//     Enc/Inputs/In/nState1 @bit 1 <-> FB Inputs Channel 2/Status/Error
//     Enc/Inputs/In/nState1 @bit 1 <-> FB Inputs Channel 1/Status/Error
//     Enc/Inputs/In/nState1 @bit 14 <-> FB Inputs Channel 2/Status/Input cycle counter
//     Enc/Inputs/In/nState1 @bit 14 <-> FB Inputs Channel 1/Status/Input cycle counter
//     Enc/Inputs/In/nState1 @bit 2 <-> FB Inputs Channel 2/Status/Ready
//     Enc/Inputs/In/nState1 @bit 2 <-> FB Inputs Channel 1/Status/Ready
//     Enc/Inputs/In/nState1 @bit 13 <-> FB Inputs Channel 2/Status/TxPDO State
//     Enc/Inputs/In/nState1 @bit 13 <-> FB Inputs Channel 1/Status/TxPDO State
//     Enc/Inputs/In/nState1 <-> FB Inputs Channel 2/Status/Warning
//     Enc/Inputs/In/nState1 <-> FB Inputs Channel 1/Status/Warning
//   (this object) <-> PLC Rail (EtherCAT)/Power (EK1200)/Fiber Coupler (EK1521-0010)/Term 123 (EK1100)/Term 73 (EK1122)/PAX-DRL-02 (EK1100)/PAX-EL7047-E17
//     Drive/Inputs/In/nState1 @bit 3 <-> STM Status/Status/Error
//     Drive/Inputs/In/nState1 @bit 7 <-> STM Status/Status/Motor stall
//     Drive/Inputs/In/nState1 @bit 5 <-> STM Status/Status/Moving negative
//     Drive/Inputs/In/nState1 @bit 4 <-> STM Status/Status/Moving positive
//     Drive/Inputs/In/nState1 @bit 1 <-> STM Status/Status/Ready
//     Drive/Inputs/In/nState1 <-> STM Status/Status/Ready to enable
//     Drive/Inputs/In/nState1 @bit 6 <-> STM Status/Status/Torque reduced
//     Drive/Inputs/In/nState1 @bit 2 <-> STM Status/Status/Warning
//     Drive/Inputs/In/nState2 @bit 3 <-> STM Status/Status/Digital input 1
//     Drive/Inputs/In/nState2 @bit 4 <-> STM Status/Status/Digital input 2
//     Drive/Inputs/In/nState2 @bit 5 <-> STM Status/Status/Sync error
//     Drive/Inputs/In/nState2 @bit 7 <-> STM Status/Status/TxPDO Toggle
//     Drive/Inputs/In/nState4 @bit 1 <-> WcState/InputToggle
//     Drive/Inputs/In/nState4 <-> WcState/WcState
//     Drive/Outputs/Out/nCtrl1 <-> STM Control/Control/Enable
//     Drive/Outputs/Out/nCtrl1 @bit 2 <-> STM Control/Control/Reduce torque
//     Drive/Outputs/Out/nCtrl1 @bit 1 <-> STM Control/Control/Reset
//     Drive/Outputs/Out/nCtrl2 @bit 3 <-> STM Control/Control/Digital output 1
//     Drive/Outputs/Out/nDataOut2[0] <-> STM Velocity/Velocity
//   (this object) <-> PLC Rail (EtherCAT)/Power (EK1200)/Fiber Coupler (EK1521-0010)/Term 123 (EK1100)/Term 73 (EK1122)/PAX-DRL-02 (EK1100)/PAX-EL7047-E15
//     Drive/Inputs/In/nState1 @bit 3 <-> STM Status/Status/Error
//     Drive/Inputs/In/nState1 @bit 7 <-> STM Status/Status/Motor stall
//     Drive/Inputs/In/nState1 @bit 5 <-> STM Status/Status/Moving negative
//     Drive/Inputs/In/nState1 @bit 4 <-> STM Status/Status/Moving positive
//     Drive/Inputs/In/nState1 @bit 1 <-> STM Status/Status/Ready
//     Drive/Inputs/In/nState1 <-> STM Status/Status/Ready to enable
//     Drive/Inputs/In/nState1 @bit 6 <-> STM Status/Status/Torque reduced
//     Drive/Inputs/In/nState1 @bit 2 <-> STM Status/Status/Warning
//     Drive/Inputs/In/nState2 @bit 3 <-> STM Status/Status/Digital input 1
//     Drive/Inputs/In/nState2 @bit 4 <-> STM Status/Status/Digital input 2
//     Drive/Inputs/In/nState2 @bit 5 <-> STM Status/Status/Sync error
//     Drive/Inputs/In/nState2 @bit 7 <-> STM Status/Status/TxPDO Toggle
//     Drive/Inputs/In/nState4 @bit 1 <-> WcState/InputToggle
//     Drive/Inputs/In/nState4 <-> WcState/WcState
//     Drive/Outputs/Out/nCtrl1 <-> STM Control/Control/Enable
//     Drive/Outputs/Out/nCtrl1 @bit 2 <-> STM Control/Control/Reduce torque
//     Drive/Outputs/Out/nCtrl1 @bit 1 <-> STM Control/Control/Reset
//     Drive/Outputs/Out/nCtrl2 @bit 3 <-> STM Control/Control/Digital output 1
//     Drive/Outputs/Out/nDataOut2[0] <-> STM Velocity/Velocity
//   (this object) <-> PLC Rail (EtherCAT)/Power (EK1200)/Fiber Coupler (EK1521-0010)/Term 123 (EK1100)/Term 73 (EK1122)/PAX-DRL-02 (EK1100)/PAX-EL5042-E13
//     Enc/Inputs/In/nComState @bit 1 <-> WcState/InputToggle
//     Enc/Inputs/In/nComState <-> WcState/WcState
//     Enc/Inputs/In/nDataIn1 <-> FB Inputs Channel 1/Position
//     Enc/Inputs/In/nState1 @bit 12 <-> FB Inputs Channel 1/Status/Diag
//     Enc/Inputs/In/nState1 @bit 1 <-> FB Inputs Channel 1/Status/Error
//     Enc/Inputs/In/nState1 @bit 14 <-> FB Inputs Channel 1/Status/Input cycle counter
//     Enc/Inputs/In/nState1 @bit 2 <-> FB Inputs Channel 1/Status/Ready
//     Enc/Inputs/In/nState1 @bit 13 <-> FB Inputs Channel 1/Status/TxPDO State
//     Enc/Inputs/In/nState1 <-> FB Inputs Channel 1/Status/Warning
//   (this object) <-> PLC Rail (EtherCAT)/Power (EK1200)/Fiber Coupler (EK1521-0010)/Term 123 (EK1100)/Term 73 (EK1122)/PAX-DRL-02 (EK1100)/PAX-EL7047-E12
//     Drive/Inputs/In/nState1 @bit 3 <-> STM Status/Status/Error
//     Drive/Inputs/In/nState1 @bit 7 <-> STM Status/Status/Motor stall
//     Drive/Inputs/In/nState1 @bit 5 <-> STM Status/Status/Moving negative
//     Drive/Inputs/In/nState1 @bit 4 <-> STM Status/Status/Moving positive
//     Drive/Inputs/In/nState1 @bit 1 <-> STM Status/Status/Ready
//     Drive/Inputs/In/nState1 <-> STM Status/Status/Ready to enable
//     Drive/Inputs/In/nState1 @bit 6 <-> STM Status/Status/Torque reduced
//     Drive/Inputs/In/nState1 @bit 2 <-> STM Status/Status/Warning
//     Drive/Inputs/In/nState2 @bit 3 <-> STM Status/Status/Digital input 1
//     Drive/Inputs/In/nState2 @bit 4 <-> STM Status/Status/Digital input 2
//     Drive/Inputs/In/nState2 @bit 5 <-> STM Status/Status/Sync error
//     Drive/Inputs/In/nState2 @bit 7 <-> STM Status/Status/TxPDO Toggle
//     Drive/Inputs/In/nState4 @bit 1 <-> WcState/InputToggle
//     Drive/Inputs/In/nState4 <-> WcState/WcState
//     Drive/Outputs/Out/nCtrl1 <-> STM Control/Control/Enable
//     Drive/Outputs/Out/nCtrl1 @bit 2 <-> STM Control/Control/Reduce torque
//     Drive/Outputs/Out/nCtrl1 @bit 1 <-> STM Control/Control/Reset
//     Drive/Outputs/Out/nCtrl2 @bit 3 <-> STM Control/Control/Digital output 1
//     Drive/Outputs/Out/nDataOut2[0] <-> STM Velocity/Velocity
//   (this object) <-> PLC Rail (EtherCAT)/Power (EK1200)/Fiber Coupler (EK1521-0010)/Term 123 (EK1100)/Term 73 (EK1122)/PAX-DRL-02 (EK1100)/PAX-EL5042-E09
//     Enc/Inputs/In/nComState @bit 1 <-> WcState/InputToggle
//     Enc/Inputs/In/nComState <-> WcState/WcState
//     Enc/Inputs/In/nDataIn1 <-> FB Inputs Channel 2/Position
//     Enc/Inputs/In/nDataIn1 <-> FB Inputs Channel 1/Position
//     Enc/Inputs/In/nState1 @bit 12 <-> FB Inputs Channel 2/Status/Diag
//     Enc/Inputs/In/nState1 @bit 12 <-> FB Inputs Channel 1/Status/Diag
//     Enc/Inputs/In/nState1 @bit 1 <-> FB Inputs Channel 2/Status/Error
//     Enc/Inputs/In/nState1 @bit 1 <-> FB Inputs Channel 1/Status/Error
//     Enc/Inputs/In/nState1 @bit 14 <-> FB Inputs Channel 2/Status/Input cycle counter
//     Enc/Inputs/In/nState1 @bit 14 <-> FB Inputs Channel 1/Status/Input cycle counter
//     Enc/Inputs/In/nState1 @bit 2 <-> FB Inputs Channel 2/Status/Ready
//     Enc/Inputs/In/nState1 @bit 2 <-> FB Inputs Channel 1/Status/Ready
//     Enc/Inputs/In/nState1 @bit 13 <-> FB Inputs Channel 2/Status/TxPDO State
//     Enc/Inputs/In/nState1 @bit 13 <-> FB Inputs Channel 1/Status/TxPDO State
//     Enc/Inputs/In/nState1 <-> FB Inputs Channel 2/Status/Warning
//     Enc/Inputs/In/nState1 <-> FB Inputs Channel 1/Status/Warning
//   (this object) <-> PLC Rail (EtherCAT)/Power (EK1200)/Fiber Coupler (EK1521-0010)/Term 123 (EK1100)/Term 73 (EK1122)/PAX-DRL-02 (EK1100)/PAX-EL7047-E10
//     Drive/Inputs/In/nState1 @bit 3 <-> STM Status/Status/Error
//     Drive/Inputs/In/nState1 @bit 7 <-> STM Status/Status/Motor stall
//     Drive/Inputs/In/nState1 @bit 5 <-> STM Status/Status/Moving negative
//     Drive/Inputs/In/nState1 @bit 4 <-> STM Status/Status/Moving positive
//     Drive/Inputs/In/nState1 @bit 1 <-> STM Status/Status/Ready
//     Drive/Inputs/In/nState1 <-> STM Status/Status/Ready to enable
//     Drive/Inputs/In/nState1 @bit 6 <-> STM Status/Status/Torque reduced
//     Drive/Inputs/In/nState1 @bit 2 <-> STM Status/Status/Warning
//     Drive/Inputs/In/nState2 @bit 3 <-> STM Status/Status/Digital input 1
//     Drive/Inputs/In/nState2 @bit 4 <-> STM Status/Status/Digital input 2
//     Drive/Inputs/In/nState2 @bit 5 <-> STM Status/Status/Sync error
//     Drive/Inputs/In/nState2 @bit 7 <-> STM Status/Status/TxPDO Toggle
//     Drive/Inputs/In/nState4 @bit 1 <-> WcState/InputToggle
//     Drive/Inputs/In/nState4 <-> WcState/WcState
//     Drive/Outputs/Out/nCtrl1 <-> STM Control/Control/Enable
//     Drive/Outputs/Out/nCtrl1 @bit 2 <-> STM Control/Control/Reduce torque
//     Drive/Outputs/Out/nCtrl1 @bit 1 <-> STM Control/Control/Reset
//     Drive/Outputs/Out/nCtrl2 @bit 3 <-> STM Control/Control/Digital output 1
//     Drive/Outputs/Out/nDataOut2[0] <-> STM Velocity/Velocity
//   (this object) <-> PLC Rail (EtherCAT)/Power (EK1200)/Fiber Coupler (EK1521-0010)/Term 123 (EK1100)/Term 73 (EK1122)/PAX-DRL-02 (EK1100)/PAX-EL7047-E08
//     Drive/Inputs/In/nState1 @bit 3 <-> STM Status/Status/Error
//     Drive/Inputs/In/nState1 @bit 7 <-> STM Status/Status/Motor stall
//     Drive/Inputs/In/nState1 @bit 5 <-> STM Status/Status/Moving negative
//     Drive/Inputs/In/nState1 @bit 4 <-> STM Status/Status/Moving positive
//     Drive/Inputs/In/nState1 @bit 1 <-> STM Status/Status/Ready
//     Drive/Inputs/In/nState1 <-> STM Status/Status/Ready to enable
//     Drive/Inputs/In/nState1 @bit 6 <-> STM Status/Status/Torque reduced
//     Drive/Inputs/In/nState1 @bit 2 <-> STM Status/Status/Warning
//     Drive/Inputs/In/nState2 @bit 3 <-> STM Status/Status/Digital input 1
//     Drive/Inputs/In/nState2 @bit 4 <-> STM Status/Status/Digital input 2
//     Drive/Inputs/In/nState2 @bit 5 <-> STM Status/Status/Sync error
//     Drive/Inputs/In/nState2 @bit 7 <-> STM Status/Status/TxPDO Toggle
//     Drive/Inputs/In/nState4 @bit 1 <-> WcState/InputToggle
//     Drive/Inputs/In/nState4 <-> WcState/WcState
//     Drive/Outputs/Out/nCtrl1 <-> STM Control/Control/Enable
//     Drive/Outputs/Out/nCtrl1 @bit 2 <-> STM Control/Control/Reduce torque
//     Drive/Outputs/Out/nCtrl1 @bit 1 <-> STM Control/Control/Reset
//     Drive/Outputs/Out/nCtrl2 @bit 3 <-> STM Control/Control/Digital output 1
//     Drive/Outputs/Out/nDataOut2[0] <-> STM Velocity/Velocity
//   (this object) <-> PLC Rail (EtherCAT)/Power (EK1200)/Fiber Coupler (EK1521-0010)/Term 123 (EK1100)/Term 73 (EK1122)/PAX-DRL-02 (EK1100)/PAX-EL5042-E05
//     Enc/Inputs/In/nComState @bit 1 <-> WcState/InputToggle
//     Enc/Inputs/In/nComState <-> WcState/WcState
//     Enc/Inputs/In/nDataIn1 <-> FB Inputs Channel 2/Position
//     Enc/Inputs/In/nDataIn1 <-> FB Inputs Channel 1/Position
//     Enc/Inputs/In/nState1 @bit 12 <-> FB Inputs Channel 2/Status/Diag
//     Enc/Inputs/In/nState1 @bit 12 <-> FB Inputs Channel 1/Status/Diag
//     Enc/Inputs/In/nState1 @bit 1 <-> FB Inputs Channel 2/Status/Error
//     Enc/Inputs/In/nState1 @bit 1 <-> FB Inputs Channel 1/Status/Error
//     Enc/Inputs/In/nState1 @bit 14 <-> FB Inputs Channel 2/Status/Input cycle counter
//     Enc/Inputs/In/nState1 @bit 14 <-> FB Inputs Channel 1/Status/Input cycle counter
//     Enc/Inputs/In/nState1 @bit 2 <-> FB Inputs Channel 2/Status/Ready
//     Enc/Inputs/In/nState1 @bit 2 <-> FB Inputs Channel 1/Status/Ready
//     Enc/Inputs/In/nState1 @bit 13 <-> FB Inputs Channel 2/Status/TxPDO State
//     Enc/Inputs/In/nState1 @bit 13 <-> FB Inputs Channel 1/Status/TxPDO State
//     Enc/Inputs/In/nState1 <-> FB Inputs Channel 2/Status/Warning
//     Enc/Inputs/In/nState1 <-> FB Inputs Channel 1/Status/Warning
//   (this object) <-> PLC Rail (EtherCAT)/Power (EK1200)/Fiber Coupler (EK1521-0010)/Term 123 (EK1100)/Term 73 (EK1122)/PAX-DRL-02 (EK1100)/PAX-EL7047-E06
//     Drive/Inputs/In/nState1 @bit 3 <-> STM Status/Status/Error
//     Drive/Inputs/In/nState1 @bit 7 <-> STM Status/Status/Motor stall
//     Drive/Inputs/In/nState1 @bit 5 <-> STM Status/Status/Moving negative
//     Drive/Inputs/In/nState1 @bit 4 <-> STM Status/Status/Moving positive
//     Drive/Inputs/In/nState1 @bit 1 <-> STM Status/Status/Ready
//     Drive/Inputs/In/nState1 <-> STM Status/Status/Ready to enable
//     Drive/Inputs/In/nState1 @bit 6 <-> STM Status/Status/Torque reduced
//     Drive/Inputs/In/nState1 @bit 2 <-> STM Status/Status/Warning
//     Drive/Inputs/In/nState2 @bit 3 <-> STM Status/Status/Digital input 1
//     Drive/Inputs/In/nState2 @bit 4 <-> STM Status/Status/Digital input 2
//     Drive/Inputs/In/nState2 @bit 5 <-> STM Status/Status/Sync error
//     Drive/Inputs/In/nState2 @bit 7 <-> STM Status/Status/TxPDO Toggle
//     Drive/Inputs/In/nState4 @bit 1 <-> WcState/InputToggle
//     Drive/Inputs/In/nState4 <-> WcState/WcState
//     Drive/Outputs/Out/nCtrl1 <-> STM Control/Control/Enable
//     Drive/Outputs/Out/nCtrl1 @bit 2 <-> STM Control/Control/Reduce torque
//     Drive/Outputs/Out/nCtrl1 @bit 1 <-> STM Control/Control/Reset
//     Drive/Outputs/Out/nCtrl2 @bit 3 <-> STM Control/Control/Digital output 1
//     Drive/Outputs/Out/nDataOut2[0] <-> STM Velocity/Velocity
//   (this object) <-> PLC Rail (EtherCAT)/Power (EK1200)/Fiber Coupler (EK1521-0010)/Term 123 (EK1100)/Term 73 (EK1122)/PAX-DRL-02 (EK1100)/PAX-EL7047-E04
//     Drive/Inputs/In/nState1 @bit 3 <-> STM Status/Status/Error
//     Drive/Inputs/In/nState1 @bit 7 <-> STM Status/Status/Motor stall
//     Drive/Inputs/In/nState1 @bit 5 <-> STM Status/Status/Moving negative
//     Drive/Inputs/In/nState1 @bit 4 <-> STM Status/Status/Moving positive
//     Drive/Inputs/In/nState1 @bit 1 <-> STM Status/Status/Ready
//     Drive/Inputs/In/nState1 <-> STM Status/Status/Ready to enable
//     Drive/Inputs/In/nState1 @bit 6 <-> STM Status/Status/Torque reduced
//     Drive/Inputs/In/nState1 @bit 2 <-> STM Status/Status/Warning
//     Drive/Inputs/In/nState2 @bit 3 <-> STM Status/Status/Digital input 1
//     Drive/Inputs/In/nState2 @bit 4 <-> STM Status/Status/Digital input 2
//     Drive/Inputs/In/nState2 @bit 5 <-> STM Status/Status/Sync error
//     Drive/Inputs/In/nState2 @bit 7 <-> STM Status/Status/TxPDO Toggle
//     Drive/Inputs/In/nState4 @bit 1 <-> WcState/InputToggle
//     Drive/Inputs/In/nState4 <-> WcState/WcState
//     Drive/Outputs/Out/nCtrl1 <-> STM Control/Control/Enable
//     Drive/Outputs/Out/nCtrl1 @bit 2 <-> STM Control/Control/Reduce torque
//     Drive/Outputs/Out/nCtrl1 @bit 1 <-> STM Control/Control/Reset
//     Drive/Outputs/Out/nCtrl2 @bit 3 <-> STM Control/Control/Digital output 1
//     Drive/Outputs/Out/nDataOut2[0] <-> STM Velocity/Velocity
//   (this object) <-> PLC Rail (EtherCAT)/Power (EK1200)/Fiber Coupler (EK1521-0010)/Term 123 (EK1100)/Term 73 (EK1122)/PAX-DRL-02 (EK1100)/PAX-EL5042-E02
//     Enc/Inputs/In/nComState @bit 1 <-> WcState/InputToggle
//     Enc/Inputs/In/nComState <-> WcState/WcState
//     Enc/Inputs/In/nDataIn1 <-> FB Inputs Channel 2/Position
//     Enc/Inputs/In/nDataIn1 <-> FB Inputs Channel 1/Position
//     Enc/Inputs/In/nState1 @bit 12 <-> FB Inputs Channel 2/Status/Diag
//     Enc/Inputs/In/nState1 @bit 12 <-> FB Inputs Channel 1/Status/Diag
//     Enc/Inputs/In/nState1 @bit 1 <-> FB Inputs Channel 2/Status/Error
//     Enc/Inputs/In/nState1 @bit 1 <-> FB Inputs Channel 1/Status/Error
//     Enc/Inputs/In/nState1 @bit 14 <-> FB Inputs Channel 2/Status/Input cycle counter
//     Enc/Inputs/In/nState1 @bit 14 <-> FB Inputs Channel 1/Status/Input cycle counter
//     Enc/Inputs/In/nState1 @bit 2 <-> FB Inputs Channel 2/Status/Ready
//     Enc/Inputs/In/nState1 @bit 2 <-> FB Inputs Channel 1/Status/Ready
//     Enc/Inputs/In/nState1 @bit 13 <-> FB Inputs Channel 2/Status/TxPDO State
//     Enc/Inputs/In/nState1 @bit 13 <-> FB Inputs Channel 1/Status/TxPDO State
//     Enc/Inputs/In/nState1 <-> FB Inputs Channel 2/Status/Warning
//     Enc/Inputs/In/nState1 <-> FB Inputs Channel 1/Status/Warning
//   (this object) <-> PLC Rail (EtherCAT)/Power (EK1200)/Fiber Coupler (EK1521-0010)/Term 123 (EK1100)/Term 73 (EK1122)/PAX-DRL-02 (EK1100)/PAX-EL7047-E03
//     Drive/Inputs/In/nState1 @bit 3 <-> STM Status/Status/Error
//     Drive/Inputs/In/nState1 @bit 7 <-> STM Status/Status/Motor stall
//     Drive/Inputs/In/nState1 @bit 5 <-> STM Status/Status/Moving negative
//     Drive/Inputs/In/nState1 @bit 4 <-> STM Status/Status/Moving positive
//     Drive/Inputs/In/nState1 @bit 1 <-> STM Status/Status/Ready
//     Drive/Inputs/In/nState1 <-> STM Status/Status/Ready to enable
//     Drive/Inputs/In/nState1 @bit 6 <-> STM Status/Status/Torque reduced
//     Drive/Inputs/In/nState1 @bit 2 <-> STM Status/Status/Warning
//     Drive/Inputs/In/nState2 @bit 3 <-> STM Status/Status/Digital input 1
//     Drive/Inputs/In/nState2 @bit 4 <-> STM Status/Status/Digital input 2
//     Drive/Inputs/In/nState2 @bit 5 <-> STM Status/Status/Sync error
//     Drive/Inputs/In/nState2 @bit 7 <-> STM Status/Status/TxPDO Toggle
//     Drive/Inputs/In/nState4 @bit 1 <-> WcState/InputToggle
//     Drive/Inputs/In/nState4 <-> WcState/WcState
//     Drive/Outputs/Out/nCtrl1 <-> STM Control/Control/Enable
//     Drive/Outputs/Out/nCtrl1 @bit 2 <-> STM Control/Control/Reduce torque
//     Drive/Outputs/Out/nCtrl1 @bit 1 <-> STM Control/Control/Reset
//     Drive/Outputs/Out/nCtrl2 @bit 3 <-> STM Control/Control/Digital output 1
//     Drive/Outputs/Out/nDataOut2[0] <-> STM Velocity/Velocity
//   (this object) <-> PLC Rail (EtherCAT)/Power (EK1200)/Fiber Coupler (EK1521-0010)/Term 123 (EK1100)/Term 73 (EK1122)/PAX-DRL-02 (EK1100)/PAX-EL7047-E01
//     Drive/Inputs/In/nState1 @bit 3 <-> STM Status/Status/Error
//     Drive/Inputs/In/nState1 @bit 7 <-> STM Status/Status/Motor stall
//     Drive/Inputs/In/nState1 @bit 5 <-> STM Status/Status/Moving negative
//     Drive/Inputs/In/nState1 @bit 4 <-> STM Status/Status/Moving positive
//     Drive/Inputs/In/nState1 @bit 1 <-> STM Status/Status/Ready
//     Drive/Inputs/In/nState1 <-> STM Status/Status/Ready to enable
//     Drive/Inputs/In/nState1 @bit 6 <-> STM Status/Status/Torque reduced
//     Drive/Inputs/In/nState1 @bit 2 <-> STM Status/Status/Warning
//     Drive/Inputs/In/nState2 @bit 3 <-> STM Status/Status/Digital input 1
//     Drive/Inputs/In/nState2 @bit 4 <-> STM Status/Status/Digital input 2
//     Drive/Inputs/In/nState2 @bit 5 <-> STM Status/Status/Sync error
//     Drive/Inputs/In/nState2 @bit 7 <-> STM Status/Status/TxPDO Toggle
//     Drive/Inputs/In/nState4 @bit 1 <-> WcState/InputToggle
//     Drive/Inputs/In/nState4 <-> WcState/WcState
//     Drive/Outputs/Out/nCtrl1 <-> STM Control/Control/Enable
//     Drive/Outputs/Out/nCtrl1 @bit 2 <-> STM Control/Control/Reduce torque
//     Drive/Outputs/Out/nCtrl1 @bit 1 <-> STM Control/Control/Reset
//     Drive/Outputs/Out/nCtrl2 @bit 3 <-> STM Control/Control/Digital output 1
//     Drive/Outputs/Out/nDataOut2[0] <-> STM Velocity/Velocity
//   kfe_rix_motion Instance <-> PLC Rail (EtherCAT)/EtherCAT Panel (EK1100)/EC E1 (EK1122)/X1 IM1K1-PPM (EK1100)/IM1K1-EL2004
//     PlcTask Outputs/Main.M1.bBrakeRelease <-> Channel 1/Output
//     PlcTask Outputs/PRG_IM1K1_PPM.fbIM1K1.fbGige.bGigePower <-> Channel 2/Output
//   kfe_rix_motion Instance <-> PLC Rail (EtherCAT)/EtherCAT Panel (EK1100)/EC E1 (EK1122)/X1 IM1K1-PPM (EK1100)/IM1K1-EL3062
//     PlcTask Inputs/PRG_IM1K1_PPM.fbIM1K1.fbPowerMeter.iVoltageINT <-> AI Standard Channel 1/Value
//   kfe_rix_motion Instance <-> PLC Rail (EtherCAT)/EtherCAT Panel (EK1100)/EC E1 (EK1122)/X1 IM1K1-PPM (EK1100)/IM1K1-EL3314
//     PlcTask Inputs/PRG_IM1K1_PPM.fbIM1K1.fbPowerMeter.fbTempSensor.bError <-> TC Inputs Channel 1/Status/Error
//     PlcTask Inputs/PRG_IM1K1_PPM.fbIM1K1.fbPowerMeter.fbTempSensor.bOverrange <-> TC Inputs Channel 1/Status/Overrange
//     PlcTask Inputs/PRG_IM1K1_PPM.fbIM1K1.fbPowerMeter.fbTempSensor.bUnderrange <-> TC Inputs Channel 1/Status/Underrange
//     PlcTask Inputs/PRG_IM1K1_PPM.fbIM1K1.fbPowerMeter.fbTempSensor.iRaw <-> TC Inputs Channel 1/Value
//     PlcTask Inputs/PRG_IM1K1_PPM.fbIM1K1.fbYagTempSensor.bError <-> TC Inputs Channel 2/Status/Error
//     PlcTask Inputs/PRG_IM1K1_PPM.fbIM1K1.fbYagTempSensor.bOverrange <-> TC Inputs Channel 2/Status/Overrange
//     PlcTask Inputs/PRG_IM1K1_PPM.fbIM1K1.fbYagTempSensor.bUnderrange <-> TC Inputs Channel 2/Status/Underrange
//     PlcTask Inputs/PRG_IM1K1_PPM.fbIM1K1.fbYagTempSensor.iRaw <-> TC Inputs Channel 2/Value
//   kfe_rix_motion Instance <-> PLC Rail (EtherCAT)/EtherCAT Panel (EK1100)/EC E1 (EK1122)/X1 IM1K1-PPM (EK1100)/IM1K1-EL4004
//     PlcTask Outputs/PRG_IM1K1_PPM.fbIM1K1.fbGige.iIlluminatorINT <-> AO Outputs Channel 1/Analog output
//   kfe_rix_motion Instance <-> PLC Rail (EtherCAT)/EtherCAT Panel (EK1100)/EC E1 (EK1122)/X1 IM1K1-PPM (EK1100)/IM1K1-EL7041
//     PlcTask Inputs/Main.M1.bLimitBackwardEnable <-> STM Status/Status/Digital input 2
//     PlcTask Inputs/Main.M1.bLimitForwardEnable <-> STM Status/Status/Digital input 1
//   kfe_rix_motion Instance <-> PLC Rail (EtherCAT)/EtherCAT Panel (EK1100)/EC E1 (EK1122)/X2 IM2K1-PPM (EK1100)/IM2K1-EL2004
//     PlcTask Outputs/Main.M2.bBrakeRelease <-> Channel 1/Output
//     PlcTask Outputs/PRG_IM2K1_PPM.fbIM2K1.fbGige.bGigePower <-> Channel 2/Output
//   kfe_rix_motion Instance <-> PLC Rail (EtherCAT)/EtherCAT Panel (EK1100)/EC E1 (EK1122)/X2 IM2K1-PPM (EK1100)/IM2K1-EL3062
//     PlcTask Inputs/PRG_IM2K1_PPM.fbIM2K1.fbPowerMeter.iVoltageINT <-> AI Standard Channel 1/Value
//   kfe_rix_motion Instance <-> PLC Rail (EtherCAT)/EtherCAT Panel (EK1100)/EC E1 (EK1122)/X2 IM2K1-PPM (EK1100)/IM2K1-EL3314
//     PlcTask Inputs/PRG_IM2K1_PPM.fbIM2K1.fbPowerMeter.fbTempSensor.bError <-> TC Inputs Channel 1/Status/Error
//     PlcTask Inputs/PRG_IM2K1_PPM.fbIM2K1.fbPowerMeter.fbTempSensor.bOverrange <-> TC Inputs Channel 1/Status/Overrange
//     PlcTask Inputs/PRG_IM2K1_PPM.fbIM2K1.fbPowerMeter.fbTempSensor.bUnderrange <-> TC Inputs Channel 1/Status/Underrange
//     PlcTask Inputs/PRG_IM2K1_PPM.fbIM2K1.fbPowerMeter.fbTempSensor.iRaw <-> TC Inputs Channel 1/Value
//     PlcTask Inputs/PRG_IM2K1_PPM.fbIM2K1.fbYagTempSensor.bError <-> TC Inputs Channel 2/Status/Error
//     PlcTask Inputs/PRG_IM2K1_PPM.fbIM2K1.fbYagTempSensor.bOverrange <-> TC Inputs Channel 2/Status/Overrange
//     PlcTask Inputs/PRG_IM2K1_PPM.fbIM2K1.fbYagTempSensor.bUnderrange <-> TC Inputs Channel 2/Status/Underrange
//     PlcTask Inputs/PRG_IM2K1_PPM.fbIM2K1.fbYagTempSensor.iRaw <-> TC Inputs Channel 2/Value
//   kfe_rix_motion Instance <-> PLC Rail (EtherCAT)/EtherCAT Panel (EK1100)/EC E1 (EK1122)/X2 IM2K1-PPM (EK1100)/IM2K1-EL4004
//     PlcTask Outputs/PRG_IM2K1_PPM.fbIM2K1.fbGige.iIlluminatorINT <-> AO Outputs Channel 1/Analog output
//   kfe_rix_motion Instance <-> PLC Rail (EtherCAT)/EtherCAT Panel (EK1100)/EC E1 (EK1122)/X2 IM2K1-PPM (EK1100)/IM2K1-EL7041
//     PlcTask Inputs/Main.M2.bLimitBackwardEnable <-> STM Status/Status/Digital input 2
//     PlcTask Inputs/Main.M2.bLimitForwardEnable <-> STM Status/Status/Digital input 1
//   kfe_rix_motion Instance <-> PLC Rail (EtherCAT)/Power (EK1200)/Fiber Coupler (EK1521-0010)/Term 123 (EK1100)/Term 124 (EK1122)/TM1K2-K2A (EK1100)/TM1K2-EL2004-E4
//     PlcTask Outputs/Main.M9.bBrakeRelease <-> Channel 1/Output
//   kfe_rix_motion Instance <-> PLC Rail (EtherCAT)/Power (EK1200)/Fiber Coupler (EK1521-0010)/Term 123 (EK1100)/Term 124 (EK1122)/TM1K2-K2A (EK1100)/TM1K2-EL3314-E5
//     PlcTask Inputs/PRG_TM1K2_ATM.fbTM1K2.fbThermoCouple1.bError <-> TC Inputs Channel 1/Status/Error
//     PlcTask Inputs/PRG_TM1K2_ATM.fbTM1K2.fbThermoCouple1.bOverrange <-> TC Inputs Channel 1/Status/Overrange
//     PlcTask Inputs/PRG_TM1K2_ATM.fbTM1K2.fbThermoCouple1.bUnderrange <-> TC Inputs Channel 1/Status/Underrange
//     PlcTask Inputs/PRG_TM1K2_ATM.fbTM1K2.fbThermoCouple1.iRaw <-> TC Inputs Channel 1/Value
//   kfe_rix_motion Instance <-> PLC Rail (EtherCAT)/Power (EK1200)/Fiber Coupler (EK1521-0010)/Term 123 (EK1100)/Term 124 (EK1122)/TM1K2-K2A (EK1100)/TM1K2-EL5042-E3
//     PlcTask Inputs/Main.M10.nRawEncoderULINT <-> FB Inputs Channel 2/Position
//     PlcTask Inputs/Main.M9.nRawEncoderULINT <-> FB Inputs Channel 1/Position
//   kfe_rix_motion Instance <-> PLC Rail (EtherCAT)/Power (EK1200)/Fiber Coupler (EK1521-0010)/Term 123 (EK1100)/Term 124 (EK1122)/TM1K2-K2A (EK1100)/TM1K2-EL7041-E1
//     PlcTask Inputs/Main.M9.bLimitBackwardEnable <-> STM Status/Status/Digital input 2
//     PlcTask Inputs/Main.M9.bLimitForwardEnable <-> STM Status/Status/Digital input 1
//   kfe_rix_motion Instance <-> PLC Rail (EtherCAT)/Power (EK1200)/Fiber Coupler (EK1521-0010)/Term 123 (EK1100)/Term 131 (EK1122)/LI2K2-K2A_OUT  (EK1100)/LI2K2-EL2004-E2
//     PlcTask Outputs/Main.M11.bBrakeRelease <-> Channel 1/Output
//   kfe_rix_motion Instance <-> PLC Rail (EtherCAT)/Power (EK1200)/Fiber Coupler (EK1521-0010)/Term 123 (EK1100)/Term 131 (EK1122)/LI2K2-K2A_OUT  (EK1100)/LI2K2-EL5042-E3
//     PlcTask Inputs/Main.M11.nRawEncoderULINT <-> FB Inputs Channel 1/Position
//   kfe_rix_motion Instance <-> PLC Rail (EtherCAT)/Power (EK1200)/Fiber Coupler (EK1521-0010)/Term 123 (EK1100)/Term 131 (EK1122)/LI2K2-K2A_OUT  (EK1100)/LI2K2-EL7041-E1
//     PlcTask Inputs/Main.M11.bLimitBackwardEnable <-> STM Status/Status/Digital input 2
//     PlcTask Inputs/Main.M11.bLimitForwardEnable <-> STM Status/Status/Digital input 1
//   kfe_rix_motion Instance <-> PLC Rail (EtherCAT)/Power (EK1200)/Fiber Coupler (EK1521-0010)/Term 123 (EK1100)/Term 131 (EK1122)/PF1K2-WFS (EK1100)/PF1K2-EL2004-E4
//     PlcTask Outputs/Main.M12.bBrakeRelease <-> Channel 1/Output
//   kfe_rix_motion Instance <-> PLC Rail (EtherCAT)/Power (EK1200)/Fiber Coupler (EK1521-0010)/Term 123 (EK1100)/Term 131 (EK1122)/PF1K2-WFS (EK1100)/PF1K2-EL3314-E5
//     PlcTask Inputs/PRG_PF1K2_WFS.fbPF1K2.fbThermoCouple1.bError <-> TC Inputs Channel 1/Status/Error
//     PlcTask Inputs/PRG_PF1K2_WFS.fbPF1K2.fbThermoCouple2.bError <-> TC Inputs Channel 2/Status/Error
//     PlcTask Inputs/PRG_PF1K2_WFS.fbPF1K2.fbThermoCouple1.bOverrange <-> TC Inputs Channel 1/Status/Overrange
//     PlcTask Inputs/PRG_PF1K2_WFS.fbPF1K2.fbThermoCouple2.bOverrange <-> TC Inputs Channel 2/Status/Overrange
//     PlcTask Inputs/PRG_PF1K2_WFS.fbPF1K2.fbThermoCouple1.bUnderrange <-> TC Inputs Channel 1/Status/Underrange
//     PlcTask Inputs/PRG_PF1K2_WFS.fbPF1K2.fbThermoCouple2.bUnderrange <-> TC Inputs Channel 2/Status/Underrange
//     PlcTask Inputs/PRG_PF1K2_WFS.fbPF1K2.fbThermoCouple1.iRaw <-> TC Inputs Channel 1/Value
//     PlcTask Inputs/PRG_PF1K2_WFS.fbPF1K2.fbThermoCouple2.iRaw <-> TC Inputs Channel 2/Value
//   kfe_rix_motion Instance <-> PLC Rail (EtherCAT)/Power (EK1200)/Fiber Coupler (EK1521-0010)/Term 123 (EK1100)/Term 131 (EK1122)/PF1K2-WFS (EK1100)/PF1K2-EL5042-E3
//     PlcTask Inputs/Main.M12.nRawEncoderULINT <-> FB Inputs Channel 2/Position
//     PlcTask Inputs/Main.M13.nRawEncoderULINT <-> FB Inputs Channel 1/Position
//   kfe_rix_motion Instance <-> PLC Rail (EtherCAT)/Power (EK1200)/Fiber Coupler (EK1521-0010)/Term 123 (EK1100)/Term 131 (EK1122)/PF1K2-WFS (EK1100)/PF1K2-EL7041-E1
//     PlcTask Inputs/Main.M12.bLimitBackwardEnable <-> STM Status/Status/Digital input 2
//     PlcTask Inputs/Main.M12.bLimitForwardEnable <-> STM Status/Status/Digital input 1
//   kfe_rix_motion Instance <-> PLC Rail (EtherCAT)/Power (EK1200)/Fiber Coupler (EK1521-0010)/Term 123 (EK1100)/Term 140 (EK1122)/IM5K2-PPM (EK1100)/IM5K2-EL2004-E3
//     PlcTask Outputs/Main.M14.bBrakeRelease <-> Channel 1/Output
//     PlcTask Outputs/PRG_IM5K2_PPM.fbIM5K2.fbGige.bGigePower <-> Channel 2/Output
//   kfe_rix_motion Instance <-> PLC Rail (EtherCAT)/Power (EK1200)/Fiber Coupler (EK1521-0010)/Term 123 (EK1100)/Term 140 (EK1122)/IM5K2-PPM (EK1100)/IM5K2-EL3052-E5
//     PlcTask Inputs/PRG_IM5K2_PPM.fbIM5K2.fbFlowMeter.iRaw <-> AI Standard Channel 1/Value
//     PlcTask Inputs/PRG_PF1K2_WFS.fbPF1K2.fbFlowMeter.iRaw <-> AI Standard Channel 1/Value
//   kfe_rix_motion Instance <-> PLC Rail (EtherCAT)/Power (EK1200)/Fiber Coupler (EK1521-0010)/Term 123 (EK1100)/Term 140 (EK1122)/IM5K2-PPM (EK1100)/IM5K2-EL3062-E6
//     PlcTask Inputs/PRG_IM5K2_PPM.fbIM5K2.fbPowerMeter.iVoltageINT <-> AI Standard Channel 1/Value
//   kfe_rix_motion Instance <-> PLC Rail (EtherCAT)/Power (EK1200)/Fiber Coupler (EK1521-0010)/Term 123 (EK1100)/Term 140 (EK1122)/IM5K2-PPM (EK1100)/IM5K2-EL3314-E4
//     PlcTask Inputs/PRG_IM5K2_PPM.fbIM5K2.fbPowerMeter.fbTempSensor.bError <-> TC Inputs Channel 1/Status/Error
//     PlcTask Inputs/PRG_IM5K2_PPM.fbIM5K2.fbPowerMeter.fbTempSensor.bOverrange <-> TC Inputs Channel 1/Status/Overrange
//     PlcTask Inputs/PRG_IM5K2_PPM.fbIM5K2.fbPowerMeter.fbTempSensor.bUnderrange <-> TC Inputs Channel 1/Status/Underrange
//     PlcTask Inputs/PRG_IM5K2_PPM.fbIM5K2.fbPowerMeter.fbTempSensor.iRaw <-> TC Inputs Channel 1/Value
//     PlcTask Inputs/PRG_IM5K2_PPM.fbIM5K2.fbYagTempSensor.bError <-> TC Inputs Channel 2/Status/Error
//     PlcTask Inputs/PRG_IM5K2_PPM.fbIM5K2.fbYagTempSensor.bOverrange <-> TC Inputs Channel 2/Status/Overrange
//     PlcTask Inputs/PRG_IM5K2_PPM.fbIM5K2.fbYagTempSensor.bUnderrange <-> TC Inputs Channel 2/Status/Underrange
//     PlcTask Inputs/PRG_IM5K2_PPM.fbIM5K2.fbYagTempSensor.iRaw <-> TC Inputs Channel 2/Value
//   kfe_rix_motion Instance <-> PLC Rail (EtherCAT)/Power (EK1200)/Fiber Coupler (EK1521-0010)/Term 123 (EK1100)/Term 140 (EK1122)/IM5K2-PPM (EK1100)/IM5K2-EL4004-E7
//     PlcTask Outputs/PRG_IM5K2_PPM.fbIM5K2.fbGige.iIlluminatorINT <-> AO Outputs Channel 1/Analog output
//   kfe_rix_motion Instance <-> PLC Rail (EtherCAT)/Power (EK1200)/Fiber Coupler (EK1521-0010)/Term 123 (EK1100)/Term 140 (EK1122)/IM5K2-PPM (EK1100)/IM5K2-EL7041-E1
//     PlcTask Inputs/Main.M14.bLimitBackwardEnable <-> STM Status/Status/Digital input 2
//     PlcTask Inputs/Main.M14.bLimitForwardEnable <-> STM Status/Status/Digital input 1
//   kfe_rix_motion Instance <-> PLC Rail (EtherCAT)/Power (EK1200)/Fiber Coupler (EK1521-0010)/Term 123 (EK1100)/Term 140 (EK1122)/TM2K2-K2B (EK1100)/TM2K2-EL2004-E4
//     PlcTask Outputs/Main.M15.bBrakeRelease <-> Channel 1/Output
//   kfe_rix_motion Instance <-> PLC Rail (EtherCAT)/Power (EK1200)/Fiber Coupler (EK1521-0010)/Term 123 (EK1100)/Term 140 (EK1122)/TM2K2-K2B (EK1100)/TM2K2-EL3052-E6
//     PlcTask Inputs/PRG_AT2K2_SOLID.fbFlowMeter.iRaw <-> AI Standard Channel 1/Value
//     PlcTask Inputs/PRG_TM2K2_ATM.fbTM2K2.fbFlowMeter.iRaw <-> AI Standard Channel 1/Value
//   kfe_rix_motion Instance <-> PLC Rail (EtherCAT)/Power (EK1200)/Fiber Coupler (EK1521-0010)/Term 123 (EK1100)/Term 140 (EK1122)/TM2K2-K2B (EK1100)/TM2K2-EL3314-E5
//     PlcTask Inputs/PRG_TM2K2_ATM.fbTM2K2.fbThermoCouple1.bError <-> TC Inputs Channel 1/Status/Error
//     PlcTask Inputs/PRG_TM2K2_ATM.fbTM2K2.fbThermoCouple1.bOverrange <-> TC Inputs Channel 1/Status/Overrange
//     PlcTask Inputs/PRG_TM2K2_ATM.fbTM2K2.fbThermoCouple1.bUnderrange <-> TC Inputs Channel 1/Status/Underrange
//     PlcTask Inputs/PRG_TM2K2_ATM.fbTM2K2.fbThermoCouple1.iRaw <-> TC Inputs Channel 1/Value
//   kfe_rix_motion Instance <-> PLC Rail (EtherCAT)/Power (EK1200)/Fiber Coupler (EK1521-0010)/Term 123 (EK1100)/Term 140 (EK1122)/TM2K2-K2B (EK1100)/TM2K2-EL5042-E3
//     PlcTask Inputs/Main.M15.nRawEncoderULINT <-> FB Inputs Channel 1/Position
//     PlcTask Inputs/Main.M16.nRawEncoderULINT <-> FB Inputs Channel 2/Position
//   kfe_rix_motion Instance <-> PLC Rail (EtherCAT)/Power (EK1200)/Fiber Coupler (EK1521-0010)/Term 123 (EK1100)/Term 140 (EK1122)/TM2K2-K2B (EK1100)/TM2K2-EL7041-E1
//     PlcTask Inputs/Main.M15.bLimitBackwardEnable <-> STM Status/Status/Digital input 2
//     PlcTask Inputs/Main.M15.bLimitForwardEnable <-> STM Status/Status/Digital input 1
//   kfe_rix_motion Instance <-> PLC Rail (EtherCAT)/Power (EK1200)/Fiber Coupler (EK1521-0010)/Term 123 (EK1100)/Term 155 (EK1122)/AT2K2-SOLID (EK1100)/AT2K2-EL3202-01
//     PlcTask Inputs/PRG_AT2K2_SOLID.fbStage4.fbRTD_1.bError <-> RTD Inputs Channel 1/Status/Error
//     PlcTask Inputs/PRG_AT2K2_SOLID.fbStage4.fbRTD_2.bError <-> RTD Inputs Channel 2/Status/Error
//     PlcTask Inputs/PRG_AT2K2_SOLID.fbStage4.fbRTD_1.bOverrange <-> RTD Inputs Channel 1/Status/Overrange
//     PlcTask Inputs/PRG_AT2K2_SOLID.fbStage4.fbRTD_2.bOverrange <-> RTD Inputs Channel 2/Status/Overrange
//     PlcTask Inputs/PRG_AT2K2_SOLID.fbStage4.fbRTD_1.bUnderrange <-> RTD Inputs Channel 1/Status/Underrange
//     PlcTask Inputs/PRG_AT2K2_SOLID.fbStage4.fbRTD_2.bUnderrange <-> RTD Inputs Channel 2/Status/Underrange
//     PlcTask Inputs/PRG_AT2K2_SOLID.fbStage4.fbRTD_1.iRaw <-> RTD Inputs Channel 1/Value
//     PlcTask Inputs/PRG_AT2K2_SOLID.fbStage4.fbRTD_2.iRaw <-> RTD Inputs Channel 2/Value
//   kfe_rix_motion Instance <-> PLC Rail (EtherCAT)/Power (EK1200)/Fiber Coupler (EK1521-0010)/Term 123 (EK1100)/Term 155 (EK1122)/AT2K2-SOLID (EK1100)/AT2K2-EL3202-02
//     PlcTask Inputs/PRG_AT2K2_SOLID.fbStage3.fbRTD_1.bError <-> RTD Inputs Channel 1/Status/Error
//     PlcTask Inputs/PRG_AT2K2_SOLID.fbStage3.fbRTD_2.bError <-> RTD Inputs Channel 2/Status/Error
//     PlcTask Inputs/PRG_AT2K2_SOLID.fbStage3.fbRTD_1.bOverrange <-> RTD Inputs Channel 1/Status/Overrange
//     PlcTask Inputs/PRG_AT2K2_SOLID.fbStage3.fbRTD_2.bOverrange <-> RTD Inputs Channel 2/Status/Overrange
//     PlcTask Inputs/PRG_AT2K2_SOLID.fbStage3.fbRTD_1.bUnderrange <-> RTD Inputs Channel 1/Status/Underrange
//     PlcTask Inputs/PRG_AT2K2_SOLID.fbStage3.fbRTD_2.bUnderrange <-> RTD Inputs Channel 2/Status/Underrange
//     PlcTask Inputs/PRG_AT2K2_SOLID.fbStage3.fbRTD_1.iRaw <-> RTD Inputs Channel 1/Value
//     PlcTask Inputs/PRG_AT2K2_SOLID.fbStage3.fbRTD_2.iRaw <-> RTD Inputs Channel 2/Value
//   kfe_rix_motion Instance <-> PLC Rail (EtherCAT)/Power (EK1200)/Fiber Coupler (EK1521-0010)/Term 123 (EK1100)/Term 155 (EK1122)/AT2K2-SOLID (EK1100)/AT2K2-EL3202-03
//     PlcTask Inputs/PRG_AT2K2_SOLID.fbStage2.fbRTD_1.bError <-> RTD Inputs Channel 1/Status/Error
//     PlcTask Inputs/PRG_AT2K2_SOLID.fbStage2.fbRTD_2.bError <-> RTD Inputs Channel 2/Status/Error
//     PlcTask Inputs/PRG_AT2K2_SOLID.fbStage2.fbRTD_1.bOverrange <-> RTD Inputs Channel 1/Status/Overrange
//     PlcTask Inputs/PRG_AT2K2_SOLID.fbStage2.fbRTD_2.bOverrange <-> RTD Inputs Channel 2/Status/Overrange
//     PlcTask Inputs/PRG_AT2K2_SOLID.fbStage2.fbRTD_1.bUnderrange <-> RTD Inputs Channel 1/Status/Underrange
//     PlcTask Inputs/PRG_AT2K2_SOLID.fbStage2.fbRTD_2.bUnderrange <-> RTD Inputs Channel 2/Status/Underrange
//     PlcTask Inputs/PRG_AT2K2_SOLID.fbStage2.fbRTD_1.iRaw <-> RTD Inputs Channel 1/Value
//     PlcTask Inputs/PRG_AT2K2_SOLID.fbStage2.fbRTD_2.iRaw <-> RTD Inputs Channel 2/Value
//   kfe_rix_motion Instance <-> PLC Rail (EtherCAT)/Power (EK1200)/Fiber Coupler (EK1521-0010)/Term 123 (EK1100)/Term 155 (EK1122)/AT2K2-SOLID (EK1100)/AT2K2-EL3202-04
//     PlcTask Inputs/PRG_AT2K2_SOLID.fbStage1.fbRTD_1.bError <-> RTD Inputs Channel 1/Status/Error
//     PlcTask Inputs/PRG_AT2K2_SOLID.fbStage1.fbRTD_2.bError <-> RTD Inputs Channel 2/Status/Error
//     PlcTask Inputs/PRG_AT2K2_SOLID.fbStage1.fbRTD_1.bOverrange <-> RTD Inputs Channel 1/Status/Overrange
//     PlcTask Inputs/PRG_AT2K2_SOLID.fbStage1.fbRTD_2.bOverrange <-> RTD Inputs Channel 2/Status/Overrange
//     PlcTask Inputs/PRG_AT2K2_SOLID.fbStage1.fbRTD_1.bUnderrange <-> RTD Inputs Channel 1/Status/Underrange
//     PlcTask Inputs/PRG_AT2K2_SOLID.fbStage1.fbRTD_2.bUnderrange <-> RTD Inputs Channel 2/Status/Underrange
//     PlcTask Inputs/PRG_AT2K2_SOLID.fbStage1.fbRTD_1.iRaw <-> RTD Inputs Channel 1/Value
//     PlcTask Inputs/PRG_AT2K2_SOLID.fbStage1.fbRTD_2.iRaw <-> RTD Inputs Channel 2/Value
//   kfe_rix_motion Instance <-> PLC Rail (EtherCAT)/Power (EK1200)/Fiber Coupler (EK1521-0010)/Term 123 (EK1100)/Term 155 (EK1122)/AT2K2-SOLID (EK1100)/AT2K2-EL5042-01
//     PlcTask Inputs/Main.M17.nRawEncoderULINT <-> FB Inputs Channel 1/Position
//     PlcTask Inputs/Main.M18.nRawEncoderULINT <-> FB Inputs Channel 2/Position
//   kfe_rix_motion Instance <-> PLC Rail (EtherCAT)/Power (EK1200)/Fiber Coupler (EK1521-0010)/Term 123 (EK1100)/Term 155 (EK1122)/AT2K2-SOLID (EK1100)/AT2K2-EL5042-02
//     PlcTask Inputs/Main.M19.nRawEncoderULINT <-> FB Inputs Channel 1/Position
//     PlcTask Inputs/Main.M20.nRawEncoderULINT <-> FB Inputs Channel 2/Position
//   kfe_rix_motion Instance <-> PLC Rail (EtherCAT)/Power (EK1200)/Fiber Coupler (EK1521-0010)/Term 123 (EK1100)/Term 155 (EK1122)/AT2K2-SOLID (EK1100)/AT2K2-EL7047-01
//     PlcTask Inputs/Main.M17.bLimitBackwardEnable <-> STM Status/Status/Digital input 2
//     PlcTask Inputs/Main.M17.bLimitForwardEnable <-> STM Status/Status/Digital input 1
//   kfe_rix_motion Instance <-> PLC Rail (EtherCAT)/Power (EK1200)/Fiber Coupler (EK1521-0010)/Term 123 (EK1100)/Term 155 (EK1122)/AT2K2-SOLID (EK1100)/AT2K2-EL7047-02
//     PlcTask Inputs/Main.M18.bLimitBackwardEnable <-> STM Status/Status/Digital input 2
//     PlcTask Inputs/Main.M18.bLimitForwardEnable <-> STM Status/Status/Digital input 1
//   kfe_rix_motion Instance <-> PLC Rail (EtherCAT)/Power (EK1200)/Fiber Coupler (EK1521-0010)/Term 123 (EK1100)/Term 155 (EK1122)/AT2K2-SOLID (EK1100)/AT2K2-EL7047-03
//     PlcTask Inputs/Main.M19.bLimitBackwardEnable <-> STM Status/Status/Digital input 2
//     PlcTask Inputs/Main.M19.bLimitForwardEnable <-> STM Status/Status/Digital input 1
//   kfe_rix_motion Instance <-> PLC Rail (EtherCAT)/Power (EK1200)/Fiber Coupler (EK1521-0010)/Term 123 (EK1100)/Term 155 (EK1122)/AT2K2-SOLID (EK1100)/AT2K2-EL7047-04
//     PlcTask Inputs/Main.M20.bLimitBackwardEnable <-> STM Status/Status/Digital input 2
//     PlcTask Inputs/Main.M20.bLimitForwardEnable <-> STM Status/Status/Digital input 1
//   kfe_rix_motion Instance <-> PLC Rail (EtherCAT)/Power (EK1200)/Fiber Coupler (EK1521-0010)/Term 123 (EK1100)/Term 155 (EK1122)/LI3K2-K2B (EK1100)/LI3K2-EL2004-E3
//     PlcTask Outputs/Main.M21.bBrakeRelease <-> Channel 1/Output
//   kfe_rix_motion Instance <-> PLC Rail (EtherCAT)/Power (EK1200)/Fiber Coupler (EK1521-0010)/Term 123 (EK1100)/Term 155 (EK1122)/LI3K2-K2B (EK1100)/LI3K2-EL5042-E2
//     PlcTask Inputs/Main.M21.nRawEncoderULINT <-> FB Inputs Channel 1/Position
//   kfe_rix_motion Instance <-> PLC Rail (EtherCAT)/Power (EK1200)/Fiber Coupler (EK1521-0010)/Term 123 (EK1100)/Term 155 (EK1122)/LI3K2-K2B (EK1100)/LI3K2-EL7041-E1
//     PlcTask Inputs/Main.M21.bLimitBackwardEnable <-> STM Status/Status/Digital input 2
//     PlcTask Inputs/Main.M21.bLimitForwardEnable <-> STM Status/Status/Digital input 1
//   kfe_rix_motion Instance <-> PLC Rail (EtherCAT)/Power (EK1200)/Fiber Coupler (EK1521-0010)/Term 123 (EK1100)/Term 156 (EK1122)/IM6K2-PPM (EK1100)/IM6K2-EL2004-E3
//     PlcTask Outputs/Main.M24.bBrakeRelease <-> Channel 1/Output
//     PlcTask Outputs/PRG_IM6K2_PPM.fbIM6K2.fbGige.bGigePower <-> Channel 2/Output
//   kfe_rix_motion Instance <-> PLC Rail (EtherCAT)/Power (EK1200)/Fiber Coupler (EK1521-0010)/Term 123 (EK1100)/Term 156 (EK1122)/IM6K2-PPM (EK1100)/IM6K2-EL3314-E4
//     PlcTask Inputs/PRG_IM6K2_PPM.fbIM6K2.fbPowerMeter.fbTempSensor.bError <-> TC Inputs Channel 1/Status/Error
//     PlcTask Inputs/PRG_IM6K2_PPM.fbIM6K2.fbPowerMeter.fbTempSensor.bOverrange <-> TC Inputs Channel 1/Status/Overrange
//     PlcTask Inputs/PRG_IM6K2_PPM.fbIM6K2.fbPowerMeter.fbTempSensor.bUnderrange <-> TC Inputs Channel 1/Status/Underrange
//     PlcTask Inputs/PRG_IM6K2_PPM.fbIM6K2.fbPowerMeter.fbTempSensor.iRaw <-> TC Inputs Channel 1/Value
//     PlcTask Inputs/PRG_IM6K2_PPM.fbIM6K2.fbYagTempSensor.bError <-> TC Inputs Channel 2/Status/Error
//     PlcTask Inputs/PRG_IM6K2_PPM.fbIM6K2.fbYagTempSensor.bOverrange <-> TC Inputs Channel 2/Status/Overrange
//     PlcTask Inputs/PRG_IM6K2_PPM.fbIM6K2.fbYagTempSensor.bUnderrange <-> TC Inputs Channel 2/Status/Underrange
//     PlcTask Inputs/PRG_IM6K2_PPM.fbIM6K2.fbYagTempSensor.iRaw <-> TC Inputs Channel 2/Value
//   kfe_rix_motion Instance <-> PLC Rail (EtherCAT)/Power (EK1200)/Fiber Coupler (EK1521-0010)/Term 123 (EK1100)/Term 156 (EK1122)/IM6K2-PPM (EK1100)/IM6K2-EL3602-E8
//     PlcTask Inputs/PRG_IM6K2_PPM.fbIM6K2.fbPowerMeter.iVoltageINT <-> AI Inputs Channel 1/Value
//   kfe_rix_motion Instance <-> PLC Rail (EtherCAT)/Power (EK1200)/Fiber Coupler (EK1521-0010)/Term 123 (EK1100)/Term 156 (EK1122)/IM6K2-PPM (EK1100)/IM6K2-EL4004-E7
//     PlcTask Outputs/PRG_IM6K2_PPM.fbIM6K2.fbGige.iIlluminatorINT <-> AO Outputs Channel 1/Analog output
//   kfe_rix_motion Instance <-> PLC Rail (EtherCAT)/Power (EK1200)/Fiber Coupler (EK1521-0010)/Term 123 (EK1100)/Term 156 (EK1122)/IM6K2-PPM (EK1100)/IM6K2-EL7041-E1
//     PlcTask Inputs/Main.M24.bLimitBackwardEnable <-> STM Status/Status/Digital input 2
//     PlcTask Inputs/Main.M24.bLimitForwardEnable <-> STM Status/Status/Digital input 1
//   kfe_rix_motion Instance <-> PLC Rail (EtherCAT)/Power (EK1200)/Fiber Coupler (EK1521-0010)/Term 123 (EK1100)/Term 156 (EK1122)/PF2K2-WFS (EK1100)/PF2K2-EL2004-E4
//     PlcTask Outputs/Main.M22.bBrakeRelease <-> Channel 1/Output
//   kfe_rix_motion Instance <-> PLC Rail (EtherCAT)/Power (EK1200)/Fiber Coupler (EK1521-0010)/Term 123 (EK1100)/Term 156 (EK1122)/PF2K2-WFS (EK1100)/PF2K2-EL3314-E5
//     PlcTask Inputs/PRG_PF2K2_WFS.fbPF2K2.fbThermoCouple1.bError <-> TC Inputs Channel 1/Status/Error
//     PlcTask Inputs/PRG_PF2K2_WFS.fbPF2K2.fbThermoCouple2.bError <-> TC Inputs Channel 2/Status/Error
//     PlcTask Inputs/PRG_PF2K2_WFS.fbPF2K2.fbThermoCouple1.bOverrange <-> TC Inputs Channel 1/Status/Overrange
//     PlcTask Inputs/PRG_PF2K2_WFS.fbPF2K2.fbThermoCouple2.bOverrange <-> TC Inputs Channel 2/Status/Overrange
//     PlcTask Inputs/PRG_PF2K2_WFS.fbPF2K2.fbThermoCouple1.bUnderrange <-> TC Inputs Channel 1/Status/Underrange
//     PlcTask Inputs/PRG_PF2K2_WFS.fbPF2K2.fbThermoCouple2.bUnderrange <-> TC Inputs Channel 2/Status/Underrange
//     PlcTask Inputs/PRG_PF2K2_WFS.fbPF2K2.fbThermoCouple1.iRaw <-> TC Inputs Channel 1/Value
//     PlcTask Inputs/PRG_PF2K2_WFS.fbPF2K2.fbThermoCouple2.iRaw <-> TC Inputs Channel 2/Value
//   kfe_rix_motion Instance <-> PLC Rail (EtherCAT)/Power (EK1200)/Fiber Coupler (EK1521-0010)/Term 123 (EK1100)/Term 156 (EK1122)/PF2K2-WFS (EK1100)/PF2K2-EL5042-E3
//     PlcTask Inputs/Main.M22.nRawEncoderULINT <-> FB Inputs Channel 2/Position
//     PlcTask Inputs/Main.M23.nRawEncoderULINT <-> FB Inputs Channel 1/Position
//   kfe_rix_motion Instance <-> PLC Rail (EtherCAT)/Power (EK1200)/Fiber Coupler (EK1521-0010)/Term 123 (EK1100)/Term 156 (EK1122)/PF2K2-WFS (EK1100)/PF2K2-EL7041-E1
//     PlcTask Inputs/Main.M22.bLimitBackwardEnable <-> STM Status/Status/Digital input 2
//     PlcTask Inputs/Main.M22.bLimitForwardEnable <-> STM Status/Status/Digital input 1
//   kfe_rix_motion Instance <-> PLC Rail (EtherCAT)/Power (EK1200)/Fiber Coupler (EK1521-0010)/Term 123 (EK1100)/Term 157 (EK1122)/AT1K2-SOLID (EK1100)/AT1K2-EL3052-E8
//     PlcTask Inputs/PRG_AT1K2_SOLID.fbFlowMeter.iRaw <-> AI Standard Channel 1/Value
//     PlcTask Inputs/PRG_TM1K2_ATM.fbTM1K2.fbFlowMeter.iRaw <-> AI Standard Channel 1/Value
//   kfe_rix_motion Instance <-> PLC Rail (EtherCAT)/Power (EK1200)/Fiber Coupler (EK1521-0010)/Term 123 (EK1100)/Term 157 (EK1122)/AT1K2-SOLID (EK1100)/AT1K2-EL3202-01
//     PlcTask Inputs/PRG_AT1K2_SOLID.fbStage1.fbRTD_1.bError <-> RTD Inputs Channel 1/Status/Error
//     PlcTask Inputs/PRG_AT1K2_SOLID.fbStage1.fbRTD_2.bError <-> RTD Inputs Channel 2/Status/Error
//     PlcTask Inputs/PRG_AT1K2_SOLID.fbStage1.fbRTD_1.bOverrange <-> RTD Inputs Channel 1/Status/Overrange
//     PlcTask Inputs/PRG_AT1K2_SOLID.fbStage1.fbRTD_2.bOverrange <-> RTD Inputs Channel 2/Status/Overrange
//     PlcTask Inputs/PRG_AT1K2_SOLID.fbStage1.fbRTD_1.bUnderrange <-> RTD Inputs Channel 1/Status/Underrange
//     PlcTask Inputs/PRG_AT1K2_SOLID.fbStage1.fbRTD_2.bUnderrange <-> RTD Inputs Channel 2/Status/Underrange
//     PlcTask Inputs/PRG_AT1K2_SOLID.fbStage1.fbRTD_1.iRaw <-> RTD Inputs Channel 1/Value
//     PlcTask Inputs/PRG_AT1K2_SOLID.fbStage1.fbRTD_2.iRaw <-> RTD Inputs Channel 2/Value
//   kfe_rix_motion Instance <-> PLC Rail (EtherCAT)/Power (EK1200)/Fiber Coupler (EK1521-0010)/Term 123 (EK1100)/Term 157 (EK1122)/AT1K2-SOLID (EK1100)/AT1K2-EL3202-02
//     PlcTask Inputs/PRG_AT1K2_SOLID.fbStage2.fbRTD_1.bError <-> RTD Inputs Channel 1/Status/Error
//     PlcTask Inputs/PRG_AT1K2_SOLID.fbStage2.fbRTD_2.bError <-> RTD Inputs Channel 2/Status/Error
//     PlcTask Inputs/PRG_AT1K2_SOLID.fbStage2.fbRTD_1.bOverrange <-> RTD Inputs Channel 1/Status/Overrange
//     PlcTask Inputs/PRG_AT1K2_SOLID.fbStage2.fbRTD_2.bOverrange <-> RTD Inputs Channel 2/Status/Overrange
//     PlcTask Inputs/PRG_AT1K2_SOLID.fbStage2.fbRTD_1.bUnderrange <-> RTD Inputs Channel 1/Status/Underrange
//     PlcTask Inputs/PRG_AT1K2_SOLID.fbStage2.fbRTD_2.bUnderrange <-> RTD Inputs Channel 2/Status/Underrange
//     PlcTask Inputs/PRG_AT1K2_SOLID.fbStage2.fbRTD_1.iRaw <-> RTD Inputs Channel 1/Value
//     PlcTask Inputs/PRG_AT1K2_SOLID.fbStage2.fbRTD_2.iRaw <-> RTD Inputs Channel 2/Value
//   kfe_rix_motion Instance <-> PLC Rail (EtherCAT)/Power (EK1200)/Fiber Coupler (EK1521-0010)/Term 123 (EK1100)/Term 157 (EK1122)/AT1K2-SOLID (EK1100)/AT1K2-EL5042-01
//     PlcTask Inputs/Main.M25.nRawEncoderULINT <-> FB Inputs Channel 1/Position
//     PlcTask Inputs/Main.M26.nRawEncoderULINT <-> FB Inputs Channel 2/Position
//   kfe_rix_motion Instance <-> PLC Rail (EtherCAT)/Power (EK1200)/Fiber Coupler (EK1521-0010)/Term 123 (EK1100)/Term 157 (EK1122)/AT1K2-SOLID (EK1100)/AT1K2-EL5042-02
//     PlcTask Inputs/Main.M27.nRawEncoderULINT <-> FB Inputs Channel 1/Position
//   kfe_rix_motion Instance <-> PLC Rail (EtherCAT)/Power (EK1200)/Fiber Coupler (EK1521-0010)/Term 123 (EK1100)/Term 157 (EK1122)/AT1K2-SOLID (EK1100)/AT1K2-EL7047-01
//     PlcTask Inputs/Main.M25.bLimitBackwardEnable <-> STM Status/Status/Digital input 2
//     PlcTask Inputs/Main.M25.bLimitForwardEnable <-> STM Status/Status/Digital input 1
//   kfe_rix_motion Instance <-> PLC Rail (EtherCAT)/Power (EK1200)/Fiber Coupler (EK1521-0010)/Term 123 (EK1100)/Term 157 (EK1122)/AT1K2-SOLID (EK1100)/AT1K2-EL7047-02
//     PlcTask Inputs/Main.M26.bLimitBackwardEnable <-> STM Status/Status/Digital input 2
//     PlcTask Inputs/Main.M26.bLimitForwardEnable <-> STM Status/Status/Digital input 1
//   kfe_rix_motion Instance <-> PLC Rail (EtherCAT)/Power (EK1200)/Fiber Coupler (EK1521-0010)/Term 123 (EK1100)/Term 73 (EK1122)/K2S18-DRL-02 (EK1100)/K2S18-DRL-02-E10 (EL3202)
//     PlcTask Inputs/PRG_AT3K2_SOLID.fbStage2.fbRTD_1.bError <-> RTD Inputs Channel 1/Status/Error
//     PlcTask Inputs/PRG_AT3K2_SOLID.fbStage2.fbRTD_2.bError <-> RTD Inputs Channel 2/Status/Error
//     PlcTask Inputs/PRG_AT3K2_SOLID.fbStage2.fbRTD_1.bOverrange <-> RTD Inputs Channel 1/Status/Overrange
//     PlcTask Inputs/PRG_AT3K2_SOLID.fbStage2.fbRTD_2.bOverrange <-> RTD Inputs Channel 2/Status/Overrange
//     PlcTask Inputs/PRG_AT3K2_SOLID.fbStage2.fbRTD_1.bUnderrange <-> RTD Inputs Channel 1/Status/Underrange
//     PlcTask Inputs/PRG_AT3K2_SOLID.fbStage2.fbRTD_2.bUnderrange <-> RTD Inputs Channel 2/Status/Underrange
//     PlcTask Inputs/PRG_AT3K2_SOLID.fbStage2.fbRTD_1.iRaw <-> RTD Inputs Channel 1/Value
//     PlcTask Inputs/PRG_AT3K2_SOLID.fbStage2.fbRTD_2.iRaw <-> RTD Inputs Channel 2/Value
//   kfe_rix_motion Instance <-> PLC Rail (EtherCAT)/Power (EK1200)/Fiber Coupler (EK1521-0010)/Term 123 (EK1100)/Term 73 (EK1122)/K2S18-DRL-02 (EK1100)/K2S18-DRL-02-E5 (EL5042)
//     PlcTask Inputs/Main.M39.nRawEncoderULINT <-> FB Inputs Channel 2/Position
//   kfe_rix_motion Instance <-> PLC Rail (EtherCAT)/Power (EK1200)/Fiber Coupler (EK1521-0010)/Term 123 (EK1100)/Term 73 (EK1122)/K2S18-DRL-02 (EK1100)/K2S18-DRL-02-E6 (EL7047)
//     PlcTask Inputs/Main.M39.bLimitBackwardEnable <-> STM Status/Status/Digital input 2
//     PlcTask Inputs/Main.M39.bLimitForwardEnable <-> STM Status/Status/Digital input 1
//   kfe_rix_motion Instance <-> PLC Rail (EtherCAT)/Power (EK1200)/Fiber Coupler (EK1521-0010)/Term 123 (EK1100)/Term 73 (EK1122)/K2S18-DRL-02 (EK1100)/K2S18-DRL-02-E7 (EL7047)
//     PlcTask Inputs/Main.M40.bLimitBackwardEnable <-> STM Status/Status/Digital input 2
//     PlcTask Inputs/Main.M40.bLimitForwardEnable <-> STM Status/Status/Digital input 1
//   kfe_rix_motion Instance <-> PLC Rail (EtherCAT)/Power (EK1200)/Fiber Coupler (EK1521-0010)/Term 123 (EK1100)/Term 73 (EK1122)/K2S18-DRL-02 (EK1100)/K2S18-DRL-02-E8 (EL5042)
//     PlcTask Inputs/Main.M40.nRawEncoderULINT <-> FB Inputs Channel 1/Position
//   kfe_rix_motion Instance <-> PLC Rail (EtherCAT)/Power (EK1200)/Fiber Coupler (EK1521-0010)/Term 123 (EK1100)/Term 73 (EK1122)/K2S18-DRL-02 (EK1100)/K2S18-DRL-02-E9 (EL3202)
//     PlcTask Inputs/PRG_AT3K2_SOLID.fbStage1.fbRTD_1.bError <-> RTD Inputs Channel 1/Status/Error
//     PlcTask Inputs/PRG_AT3K2_SOLID.fbStage1.fbRTD_2.bError <-> RTD Inputs Channel 2/Status/Error
//     PlcTask Inputs/PRG_AT3K2_SOLID.fbStage1.fbRTD_1.bOverrange <-> RTD Inputs Channel 1/Status/Overrange
//     PlcTask Inputs/PRG_AT3K2_SOLID.fbStage1.fbRTD_2.bOverrange <-> RTD Inputs Channel 2/Status/Overrange
//     PlcTask Inputs/PRG_AT3K2_SOLID.fbStage1.fbRTD_1.bUnderrange <-> RTD Inputs Channel 1/Status/Underrange
//     PlcTask Inputs/PRG_AT3K2_SOLID.fbStage1.fbRTD_2.bUnderrange <-> RTD Inputs Channel 2/Status/Underrange
//     PlcTask Inputs/PRG_AT3K2_SOLID.fbStage1.fbRTD_1.iRaw <-> RTD Inputs Channel 1/Value
//     PlcTask Inputs/PRG_AT3K2_SOLID.fbStage1.fbRTD_2.iRaw <-> RTD Inputs Channel 2/Value
//   kfe_rix_motion Instance <-> PLC Rail (EtherCAT)/Power (EK1200)/Fiber Coupler (EK1521-0010)/Term 123 (EK1100)/Term 73 (EK1122)/K2S18-DRL-03 (EK1100)/K2S18-DRL-03-E7 (EL7047)
//     PlcTask Inputs/Main.M38.bLimitBackwardEnable <-> STM Status/Status/Digital input 2
//     PlcTask Inputs/Main.M38.bLimitForwardEnable <-> STM Status/Status/Digital input 1
//   kfe_rix_motion Instance <-> PLC Rail (EtherCAT)/Power (EK1200)/Fiber Coupler (EK1521-0010)/Term 123 (EK1100)/Term 73 (EK1122)/K2S18-DRL-03 (EK1100)/K2S18-DRL-03-E8 (EL5112)
//     PlcTask Inputs/Main.M38.nRawEncoderULINT <-> ENC Status Channel 1/Counter value
//   kfe_rix_motion Instance <-> PLC Rail (EtherCAT)/Power (EK1200)/Fiber Coupler (EK1521-0010)/Term 123 (EK1100)/Term 73 (EK1122)/PAX-DRL-02 (EK1100)/PAX-EL2004-E07
//     PlcTask Outputs/Main.M31.bBrakeRelease <-> Channel 1/Output
//   kfe_rix_motion Instance <-> PLC Rail (EtherCAT)/Power (EK1200)/Fiber Coupler (EK1521-0010)/Term 123 (EK1100)/Term 73 (EK1122)/PAX-DRL-02 (EK1100)/PAX-EL5042-E02
//     PlcTask Inputs/Main.M28.nRawEncoderULINT <-> FB Inputs Channel 1/Position
//     PlcTask Inputs/Main.M29.nRawEncoderULINT <-> FB Inputs Channel 2/Position
//   kfe_rix_motion Instance <-> PLC Rail (EtherCAT)/Power (EK1200)/Fiber Coupler (EK1521-0010)/Term 123 (EK1100)/Term 73 (EK1122)/PAX-DRL-02 (EK1100)/PAX-EL5042-E05
//     PlcTask Inputs/Main.M30.nRawEncoderULINT <-> FB Inputs Channel 1/Position
//     PlcTask Inputs/Main.M31.nRawEncoderULINT <-> FB Inputs Channel 2/Position
//   kfe_rix_motion Instance <-> PLC Rail (EtherCAT)/Power (EK1200)/Fiber Coupler (EK1521-0010)/Term 123 (EK1100)/Term 73 (EK1122)/PAX-DRL-02 (EK1100)/PAX-EL5042-E09
//     PlcTask Inputs/Main.M32.nRawEncoderULINT <-> FB Inputs Channel 1/Position
//     PlcTask Inputs/Main.M33.nRawEncoderULINT <-> FB Inputs Channel 2/Position
//   kfe_rix_motion Instance <-> PLC Rail (EtherCAT)/Power (EK1200)/Fiber Coupler (EK1521-0010)/Term 123 (EK1100)/Term 73 (EK1122)/PAX-DRL-02 (EK1100)/PAX-EL5042-E13
//     PlcTask Inputs/Main.M34.nRawEncoderULINT <-> FB Inputs Channel 1/Position
//     PlcTask Inputs/Main.M35.nRawEncoderULINT <-> FB Inputs Channel 2/Position
//   kfe_rix_motion Instance <-> PLC Rail (EtherCAT)/Power (EK1200)/Fiber Coupler (EK1521-0010)/Term 123 (EK1100)/Term 73 (EK1122)/PAX-DRL-02 (EK1100)/PAX-EL5042-E16
//     PlcTask Inputs/Main.M36.nRawEncoderULINT <-> FB Inputs Channel 1/Position
//     PlcTask Inputs/Main.M37.nRawEncoderULINT <-> FB Inputs Channel 2/Position
//   kfe_rix_motion Instance <-> PLC Rail (EtherCAT)/Power (EK1200)/Fiber Coupler (EK1521-0010)/Term 123 (EK1100)/Term 73 (EK1122)/PAX-DRL-02 (EK1100)/PAX-EL7047-E01
//     PlcTask Inputs/Main.M28.bLimitBackwardEnable <-> STM Status/Status/Digital input 2
//     PlcTask Inputs/Main.M28.bLimitForwardEnable <-> STM Status/Status/Digital input 1
//   kfe_rix_motion Instance <-> PLC Rail (EtherCAT)/Power (EK1200)/Fiber Coupler (EK1521-0010)/Term 123 (EK1100)/Term 73 (EK1122)/PAX-DRL-02 (EK1100)/PAX-EL7047-E03
//     PlcTask Inputs/Main.M29.bLimitBackwardEnable <-> STM Status/Status/Digital input 2
//     PlcTask Inputs/Main.M29.bLimitForwardEnable <-> STM Status/Status/Digital input 1
//   kfe_rix_motion Instance <-> PLC Rail (EtherCAT)/Power (EK1200)/Fiber Coupler (EK1521-0010)/Term 123 (EK1100)/Term 73 (EK1122)/PAX-DRL-02 (EK1100)/PAX-EL7047-E04
//     PlcTask Inputs/Main.M30.bLimitBackwardEnable <-> STM Status/Status/Digital input 2
//     PlcTask Inputs/Main.M30.bLimitForwardEnable <-> STM Status/Status/Digital input 1
//   kfe_rix_motion Instance <-> PLC Rail (EtherCAT)/Power (EK1200)/Fiber Coupler (EK1521-0010)/Term 123 (EK1100)/Term 73 (EK1122)/PAX-DRL-02 (EK1100)/PAX-EL7047-E06
//     PlcTask Inputs/Main.M31.bLimitBackwardEnable <-> STM Status/Status/Digital input 1
//     PlcTask Inputs/Main.M31.bLimitForwardEnable <-> STM Status/Status/Digital input 2
//   kfe_rix_motion Instance <-> PLC Rail (EtherCAT)/Power (EK1200)/Fiber Coupler (EK1521-0010)/Term 123 (EK1100)/Term 73 (EK1122)/PAX-DRL-02 (EK1100)/PAX-EL7047-E08
//     PlcTask Inputs/Main.M32.bLimitBackwardEnable <-> STM Status/Status/Digital input 1
//     PlcTask Inputs/Main.M32.bLimitForwardEnable <-> STM Status/Status/Digital input 2
//   kfe_rix_motion Instance <-> PLC Rail (EtherCAT)/Power (EK1200)/Fiber Coupler (EK1521-0010)/Term 123 (EK1100)/Term 73 (EK1122)/PAX-DRL-02 (EK1100)/PAX-EL7047-E10
//     PlcTask Inputs/Main.M33.bLimitBackwardEnable <-> STM Status/Status/Digital input 1
//     PlcTask Inputs/Main.M33.bLimitForwardEnable <-> STM Status/Status/Digital input 2
//   kfe_rix_motion Instance <-> PLC Rail (EtherCAT)/Power (EK1200)/Fiber Coupler (EK1521-0010)/Term 123 (EK1100)/Term 73 (EK1122)/PAX-DRL-02 (EK1100)/PAX-EL7047-E12
//     PlcTask Inputs/Main.M34.bLimitBackwardEnable <-> STM Status/Status/Digital input 2
//     PlcTask Inputs/Main.M34.bLimitForwardEnable <-> STM Status/Status/Digital input 1
//   kfe_rix_motion Instance <-> PLC Rail (EtherCAT)/Power (EK1200)/Fiber Coupler (EK1521-0010)/Term 123 (EK1100)/Term 73 (EK1122)/PAX-DRL-02 (EK1100)/PAX-EL7047-E14
//     PlcTask Inputs/Main.M35.bLimitBackwardEnable <-> STM Status/Status/Digital input 2
//     PlcTask Inputs/Main.M35.bLimitForwardEnable <-> STM Status/Status/Digital input 1
//   kfe_rix_motion Instance <-> PLC Rail (EtherCAT)/Power (EK1200)/Fiber Coupler (EK1521-0010)/Term 123 (EK1100)/Term 73 (EK1122)/PAX-DRL-02 (EK1100)/PAX-EL7047-E15
//     PlcTask Inputs/Main.M36.bLimitBackwardEnable <-> STM Status/Status/Digital input 2
//     PlcTask Inputs/Main.M36.bLimitForwardEnable <-> STM Status/Status/Digital input 1
//   kfe_rix_motion Instance <-> PLC Rail (EtherCAT)/Power (EK1200)/Fiber Coupler (EK1521-0010)/Term 123 (EK1100)/Term 73 (EK1122)/PAX-DRL-02 (EK1100)/PAX-EL7047-E17
//     PlcTask Inputs/Main.M37.bLimitBackwardEnable <-> STM Status/Status/Digital input 2
//     PlcTask Inputs/Main.M37.bLimitForwardEnable <-> STM Status/Status/Digital input 1
//   kfe_rix_motion Instance <-> PLC Rail (EtherCAT)/Power (EK1200)/Fiber Coupler (EK1521-0010)/Term 34 (EK1501-0010)/Term 39 (EK1122)/AL1K2-L2SI (EK1100)/AL1K2-EL2004-E3
//     PlcTask Outputs/Main.M5.bBrakeRelease <-> Channel 1/Output
//   kfe_rix_motion Instance <-> PLC Rail (EtherCAT)/Power (EK1200)/Fiber Coupler (EK1521-0010)/Term 34 (EK1501-0010)/Term 39 (EK1122)/AL1K2-L2SI (EK1100)/AL1K2-EL4004-E4
//     PlcTask Outputs/PRG_AL1K2_L2SI.fbAL1K2.fbLaser.iLaserINT <-> AO Outputs Channel 1/Analog output
//     PlcTask Outputs/PRG_AL1K2_L2SI.fbAL1K2.fbLaser.iShutdownINT <-> AO Outputs Channel 2/Analog output
//   kfe_rix_motion Instance <-> PLC Rail (EtherCAT)/Power (EK1200)/Fiber Coupler (EK1521-0010)/Term 34 (EK1501-0010)/Term 39 (EK1122)/AL1K2-L2SI (EK1100)/AL1K2-EL5042-E2
//     PlcTask Inputs/Main.M5.nRawEncoderULINT <-> FB Inputs Channel 1/Position
//   kfe_rix_motion Instance <-> PLC Rail (EtherCAT)/Power (EK1200)/Fiber Coupler (EK1521-0010)/Term 34 (EK1501-0010)/Term 39 (EK1122)/AL1K2-L2SI (EK1100)/AL1K2-EL7041-E1
//     PlcTask Inputs/Main.M5.bLimitBackwardEnable <-> STM Status/Status/Digital input 2
//     PlcTask Inputs/Main.M5.bLimitForwardEnable <-> STM Status/Status/Digital input 1
//   kfe_rix_motion Instance <-> PLC Rail (EtherCAT)/Power (EK1200)/Fiber Coupler (EK1521-0010)/Term 34 (EK1501-0010)/Term 39 (EK1122)/IM1K2-PPM (EK1100)/IM1K2-EL2004-E3
//     PlcTask Outputs/Main.M4.bBrakeRelease <-> Channel 1/Output
//     PlcTask Outputs/PRG_IM1K2_PPM.fbIM1K2.fbGige.bGigePower <-> Channel 2/Output
//   kfe_rix_motion Instance <-> PLC Rail (EtherCAT)/Power (EK1200)/Fiber Coupler (EK1521-0010)/Term 34 (EK1501-0010)/Term 39 (EK1122)/IM1K2-PPM (EK1100)/IM1K2-EL3052-E5
//     PlcTask Inputs/PRG_IM{1..4}K2_PPM.fbIM{1..4}K2.fbFlowMeter.iRaw <-> AI Standard Channel 1/Value  (4 links)
//   kfe_rix_motion Instance <-> PLC Rail (EtherCAT)/Power (EK1200)/Fiber Coupler (EK1521-0010)/Term 34 (EK1501-0010)/Term 39 (EK1122)/IM1K2-PPM (EK1100)/IM1K2-EL3062-E6
//     PlcTask Inputs/PRG_IM1K2_PPM.fbIM1K2.fbPowerMeter.iVoltageINT <-> AI Standard Channel 1/Value
//   kfe_rix_motion Instance <-> PLC Rail (EtherCAT)/Power (EK1200)/Fiber Coupler (EK1521-0010)/Term 34 (EK1501-0010)/Term 39 (EK1122)/IM1K2-PPM (EK1100)/IM1K2-EL3314-E4
//     PlcTask Inputs/PRG_IM1K2_PPM.fbIM1K2.fbPowerMeter.fbTempSensor.bError <-> TC Inputs Channel 1/Status/Error
//     PlcTask Inputs/PRG_IM1K2_PPM.fbIM1K2.fbPowerMeter.fbTempSensor.bOverrange <-> TC Inputs Channel 1/Status/Overrange
//     PlcTask Inputs/PRG_IM1K2_PPM.fbIM1K2.fbPowerMeter.fbTempSensor.bUnderrange <-> TC Inputs Channel 1/Status/Underrange
//     PlcTask Inputs/PRG_IM1K2_PPM.fbIM1K2.fbPowerMeter.fbTempSensor.iRaw <-> TC Inputs Channel 1/Value
//     PlcTask Inputs/PRG_IM1K2_PPM.fbIM1K2.fbYagTempSensor.bError <-> TC Inputs Channel 2/Status/Error
//     PlcTask Inputs/PRG_IM1K2_PPM.fbIM1K2.fbYagTempSensor.bOverrange <-> TC Inputs Channel 2/Status/Overrange
//     PlcTask Inputs/PRG_IM1K2_PPM.fbIM1K2.fbYagTempSensor.bUnderrange <-> TC Inputs Channel 2/Status/Underrange
//     PlcTask Inputs/PRG_IM1K2_PPM.fbIM1K2.fbYagTempSensor.iRaw <-> TC Inputs Channel 2/Value
//   kfe_rix_motion Instance <-> PLC Rail (EtherCAT)/Power (EK1200)/Fiber Coupler (EK1521-0010)/Term 34 (EK1501-0010)/Term 39 (EK1122)/IM1K2-PPM (EK1100)/IM1K2-EL4004-E7
//     PlcTask Outputs/PRG_IM1K2_PPM.fbIM1K2.fbGige.iIlluminatorINT <-> AO Outputs Channel 1/Analog output
//   kfe_rix_motion Instance <-> PLC Rail (EtherCAT)/Power (EK1200)/Fiber Coupler (EK1521-0010)/Term 34 (EK1501-0010)/Term 39 (EK1122)/IM1K2-PPM (EK1100)/IM1K2-EL7041-E1
//     PlcTask Inputs/Main.M4.bLimitBackwardEnable <-> STM Status/Status/Digital input 2
//     PlcTask Inputs/Main.M4.bLimitForwardEnable <-> STM Status/Status/Digital input 1
//   kfe_rix_motion Instance <-> PLC Rail (EtherCAT)/Power (EK1200)/Fiber Coupler (EK1521-0010)/Term 34 (EK1501-0010)/Term 49 (EK1122)/IM2K2-PPM (EK1100)/IM2K2-EL2004-E3
//     PlcTask Outputs/Main.M6.bBrakeRelease <-> Channel 1/Output
//     PlcTask Outputs/PRG_IM2K2_PPM.fbIM2K2.fbGige.bGigePower <-> Channel 2/Output
//   kfe_rix_motion Instance <-> PLC Rail (EtherCAT)/Power (EK1200)/Fiber Coupler (EK1521-0010)/Term 34 (EK1501-0010)/Term 49 (EK1122)/IM2K2-PPM (EK1100)/IM2K2-EL3062-E6
//     PlcTask Inputs/PRG_IM2K2_PPM.fbIM2K2.fbPowerMeter.iVoltageINT <-> AI Standard Channel 1/Value
//   kfe_rix_motion Instance <-> PLC Rail (EtherCAT)/Power (EK1200)/Fiber Coupler (EK1521-0010)/Term 34 (EK1501-0010)/Term 49 (EK1122)/IM2K2-PPM (EK1100)/IM2K2-EL3314-E4
//     PlcTask Inputs/PRG_IM2K2_PPM.fbIM2K2.fbPowerMeter.fbTempSensor.bError <-> TC Inputs Channel 1/Status/Error
//     PlcTask Inputs/PRG_IM2K2_PPM.fbIM2K2.fbPowerMeter.fbTempSensor.bOverrange <-> TC Inputs Channel 1/Status/Overrange
//     PlcTask Inputs/PRG_IM2K2_PPM.fbIM2K2.fbPowerMeter.fbTempSensor.bUnderrange <-> TC Inputs Channel 1/Status/Underrange
//     PlcTask Inputs/PRG_IM2K2_PPM.fbIM2K2.fbPowerMeter.fbTempSensor.iRaw <-> TC Inputs Channel 1/Value
//     PlcTask Inputs/PRG_IM2K2_PPM.fbIM2K2.fbYagTempSensor.bError <-> TC Inputs Channel 2/Status/Error
//     PlcTask Inputs/PRG_IM2K2_PPM.fbIM2K2.fbYagTempSensor.bOverrange <-> TC Inputs Channel 2/Status/Overrange
//     PlcTask Inputs/PRG_IM2K2_PPM.fbIM2K2.fbYagTempSensor.bUnderrange <-> TC Inputs Channel 2/Status/Underrange
//     PlcTask Inputs/PRG_IM2K2_PPM.fbIM2K2.fbYagTempSensor.iRaw <-> TC Inputs Channel 2/Value
//   kfe_rix_motion Instance <-> PLC Rail (EtherCAT)/Power (EK1200)/Fiber Coupler (EK1521-0010)/Term 34 (EK1501-0010)/Term 49 (EK1122)/IM2K2-PPM (EK1100)/IM2K2-EL4004-E7
//     PlcTask Outputs/PRG_IM2K2_PPM.fbIM2K2.fbGige.iIlluminatorINT <-> AO Outputs Channel 1/Analog output
//   kfe_rix_motion Instance <-> PLC Rail (EtherCAT)/Power (EK1200)/Fiber Coupler (EK1521-0010)/Term 34 (EK1501-0010)/Term 49 (EK1122)/IM2K2-PPM (EK1100)/IM2K2-EL7041-E1
//     PlcTask Inputs/Main.M6.bLimitBackwardEnable <-> STM Status/Status/Digital input 2
//     PlcTask Inputs/Main.M6.bLimitForwardEnable <-> STM Status/Status/Digital input 1
//   kfe_rix_motion Instance <-> PLC Rail (EtherCAT)/Power (EK1200)/Fiber Coupler (EK1521-0010)/Term 34 (EK1501-0010)/Term 50 (EK1122)/IM3K2-PPM (EK1100)/IM3K2-EL2004-E3
//     PlcTask Outputs/Main.M7.bBrakeRelease <-> Channel 1/Output
//     PlcTask Outputs/PRG_IM3K2_PPM.fbIM3K2.fbGige.bGigePower <-> Channel 2/Output
//   kfe_rix_motion Instance <-> PLC Rail (EtherCAT)/Power (EK1200)/Fiber Coupler (EK1521-0010)/Term 34 (EK1501-0010)/Term 50 (EK1122)/IM3K2-PPM (EK1100)/IM3K2-EL3062-E6
//     PlcTask Inputs/PRG_IM3K2_PPM.fbIM3K2.fbPowerMeter.iVoltageINT <-> AI Standard Channel 1/Value
//   kfe_rix_motion Instance <-> PLC Rail (EtherCAT)/Power (EK1200)/Fiber Coupler (EK1521-0010)/Term 34 (EK1501-0010)/Term 50 (EK1122)/IM3K2-PPM (EK1100)/IM3K2-EL3314-E4
//     PlcTask Inputs/PRG_IM3K2_PPM.fbIM3K2.fbPowerMeter.fbTempSensor.bError <-> TC Inputs Channel 1/Status/Error
//     PlcTask Inputs/PRG_IM3K2_PPM.fbIM3K2.fbPowerMeter.fbTempSensor.bOverrange <-> TC Inputs Channel 1/Status/Overrange
//     PlcTask Inputs/PRG_IM3K2_PPM.fbIM3K2.fbPowerMeter.fbTempSensor.bUnderrange <-> TC Inputs Channel 1/Status/Underrange
//     PlcTask Inputs/PRG_IM3K2_PPM.fbIM3K2.fbPowerMeter.fbTempSensor.iRaw <-> TC Inputs Channel 1/Value
//     PlcTask Inputs/PRG_IM3K2_PPM.fbIM3K2.fbYagTempSensor.bError <-> TC Inputs Channel 2/Status/Error
//     PlcTask Inputs/PRG_IM3K2_PPM.fbIM3K2.fbYagTempSensor.bOverrange <-> TC Inputs Channel 2/Status/Overrange
//     PlcTask Inputs/PRG_IM3K2_PPM.fbIM3K2.fbYagTempSensor.bUnderrange <-> TC Inputs Channel 2/Status/Underrange
//     PlcTask Inputs/PRG_IM3K2_PPM.fbIM3K2.fbYagTempSensor.iRaw <-> TC Inputs Channel 2/Value
//   kfe_rix_motion Instance <-> PLC Rail (EtherCAT)/Power (EK1200)/Fiber Coupler (EK1521-0010)/Term 34 (EK1501-0010)/Term 50 (EK1122)/IM3K2-PPM (EK1100)/IM3K2-EL4004-E7
//     PlcTask Outputs/PRG_IM3K2_PPM.fbIM3K2.fbGige.iIlluminatorINT <-> AO Outputs Channel 1/Analog output
//   kfe_rix_motion Instance <-> PLC Rail (EtherCAT)/Power (EK1200)/Fiber Coupler (EK1521-0010)/Term 34 (EK1501-0010)/Term 50 (EK1122)/IM3K2-PPM (EK1100)/IM3K2-EL7041-E1
//     PlcTask Inputs/Main.M7.bLimitBackwardEnable <-> STM Status/Status/Digital input 2
//     PlcTask Inputs/Main.M7.bLimitForwardEnable <-> STM Status/Status/Digital input 1
//   kfe_rix_motion Instance <-> PLC Rail (EtherCAT)/Power (EK1200)/Fiber Coupler (EK1521-0010)/Term 34 (EK1501-0010)/Term 50 (EK1122)/IM4K2-PPM (EK1100)/IM4K2-EL2004-E3
//     PlcTask Outputs/Main.M8.bBrakeRelease <-> Channel 1/Output
//     PlcTask Outputs/PRG_IM4K2_PPM.fbIM4K2.fbGige.bGigePower <-> Channel 2/Output
//   kfe_rix_motion Instance <-> PLC Rail (EtherCAT)/Power (EK1200)/Fiber Coupler (EK1521-0010)/Term 34 (EK1501-0010)/Term 50 (EK1122)/IM4K2-PPM (EK1100)/IM4K2-EL3314-E4
//     PlcTask Inputs/PRG_IM4K2_PPM.fbIM4K2.fbPowerMeter.fbTempSensor.bError <-> TC Inputs Channel 1/Status/Error
//     PlcTask Inputs/PRG_IM4K2_PPM.fbIM4K2.fbPowerMeter.fbTempSensor.bOverrange <-> TC Inputs Channel 1/Status/Overrange
//     PlcTask Inputs/PRG_IM4K2_PPM.fbIM4K2.fbPowerMeter.fbTempSensor.bUnderrange <-> TC Inputs Channel 1/Status/Underrange
//     PlcTask Inputs/PRG_IM4K2_PPM.fbIM4K2.fbPowerMeter.fbTempSensor.iRaw <-> TC Inputs Channel 1/Value
//     PlcTask Inputs/PRG_IM4K2_PPM.fbIM4K2.fbYagTempSensor.bError <-> TC Inputs Channel 2/Status/Error
//     PlcTask Inputs/PRG_IM4K2_PPM.fbIM4K2.fbYagTempSensor.bOverrange <-> TC Inputs Channel 2/Status/Overrange
//     PlcTask Inputs/PRG_IM4K2_PPM.fbIM4K2.fbYagTempSensor.bUnderrange <-> TC Inputs Channel 2/Status/Underrange
//     PlcTask Inputs/PRG_IM4K2_PPM.fbIM4K2.fbYagTempSensor.iRaw <-> TC Inputs Channel 2/Value
//   kfe_rix_motion Instance <-> PLC Rail (EtherCAT)/Power (EK1200)/Fiber Coupler (EK1521-0010)/Term 34 (EK1501-0010)/Term 50 (EK1122)/IM4K2-PPM (EK1100)/IM4K2-EL3602-0002-E8
//     PlcTask Inputs/PRG_IM4K2_PPM.fbIM4K2.fbPowerMeter.iVoltageINT <-> AI Inputs Channel 1/Value
//   kfe_rix_motion Instance <-> PLC Rail (EtherCAT)/Power (EK1200)/Fiber Coupler (EK1521-0010)/Term 34 (EK1501-0010)/Term 50 (EK1122)/IM4K2-PPM (EK1100)/IM4K2-EL4004-E7
//     PlcTask Outputs/PRG_IM4K2_PPM.fbIM4K2.fbGige.iIlluminatorINT <-> AO Outputs Channel 1/Analog output
//   kfe_rix_motion Instance <-> PLC Rail (EtherCAT)/Power (EK1200)/Fiber Coupler (EK1521-0010)/Term 34 (EK1501-0010)/Term 50 (EK1122)/IM4K2-PPM (EK1100)/IM4K2-EL7041-E1
//     PlcTask Inputs/Main.M8.bLimitBackwardEnable <-> STM Status/Status/Digital input 2
//     PlcTask Inputs/Main.M8.bLimitForwardEnable <-> STM Status/Status/Digital input 1
//   kfe_rix_motion Instance <-> PLC Rail (EtherCAT)/Power (EK1200)/PMPS_FFO
//     PlcTask Outputs/GVL.fbFastFaultOutput1.q_xFastFaultOut <-> Channel 1/Output
//     PlcTask Outputs/GVL.fbFastFaultOutput2.q_xFastFaultOut <-> Channel 2/Output
//   kfe_rix_motion Instance <-> PLC Rail (EtherCAT)/Power (EK1200)/PMPS_PRE
//     PlcTask Inputs/PRG_3_PMPS_POST.fbArbiterIO.i_stCurrentBP <-> IO Inputs/CurrentBP
//     PlcTask Inputs/PRG_3_PMPS_POST.fbArbiterIO.xTxPDO_state <-> SYNC Inputs/TxPDO state
//     PlcTask Inputs/PRG_3_PMPS_POST.fbArbiterIO.xTxPDO_toggle <-> SYNC Inputs/TxPDO toggle
//     PlcTask Outputs/PRG_3_PMPS_POST.fbArbiterIO.q_stRequestedBP <-> IO Outputs/RequestedBP
//   kfe_rix_motion Instance <-> NC-Task 1 SAF/Axes/Axis 1 IM1K1-PPM-MMS
//     PlcTask Inputs/Main.M1.Axis.NcToPlc <-> Outputs/ToPlc
//     PlcTask Outputs/Main.M1.Axis.PlcToNc <-> Inputs/FromPlc
//   kfe_rix_motion Instance <-> NC-Task 1 SAF/Axes/Axis 10 TM1K2-MMS-X
//     PlcTask Inputs/Main.M10.Axis.NcToPlc <-> Outputs/ToPlc
//     PlcTask Outputs/Main.M10.Axis.PlcToNc <-> Inputs/FromPlc
//   kfe_rix_motion Instance <-> NC-Task 1 SAF/Axes/Axis 11 LI2K2-K2A_OUT-MMS
//     PlcTask Inputs/Main.M11.Axis.NcToPlc <-> Outputs/ToPlc
//     PlcTask Outputs/Main.M11.Axis.PlcToNc <-> Inputs/FromPlc
//   kfe_rix_motion Instance <-> NC-Task 1 SAF/Axes/Axis 12 PF1K2-WFS-MMS-Y
//     PlcTask Inputs/Main.M12.Axis.NcToPlc <-> Outputs/ToPlc
//     PlcTask Outputs/Main.M12.Axis.PlcToNc <-> Inputs/FromPlc
//   kfe_rix_motion Instance <-> NC-Task 1 SAF/Axes/Axis 13 PF1K2-WFS-MMS-Z
//     PlcTask Inputs/Main.M13.Axis.NcToPlc <-> Outputs/ToPlc
//     PlcTask Outputs/Main.M13.Axis.PlcToNc <-> Inputs/FromPlc
//   kfe_rix_motion Instance <-> NC-Task 1 SAF/Axes/Axis 14 IM5K2-PPM-MMS
//     PlcTask Inputs/Main.M14.Axis.NcToPlc <-> Outputs/ToPlc
//     PlcTask Outputs/Main.M14.Axis.PlcToNc <-> Inputs/FromPlc
//   kfe_rix_motion Instance <-> NC-Task 1 SAF/Axes/Axis 15 TM2K2-MMS-Y
//     PlcTask Inputs/Main.M15.Axis.NcToPlc <-> Outputs/ToPlc
//     PlcTask Outputs/Main.M15.Axis.PlcToNc <-> Inputs/FromPlc
//   kfe_rix_motion Instance <-> NC-Task 1 SAF/Axes/Axis 16 TM2K2-MMS-X
//     PlcTask Inputs/Main.M16.Axis.NcToPlc <-> Outputs/ToPlc
//     PlcTask Outputs/Main.M16.Axis.PlcToNc <-> Inputs/FromPlc
//   kfe_rix_motion Instance <-> NC-Task 1 SAF/Axes/Axis 17 AT2K2-SOLID-MMS-01
//     PlcTask Inputs/Main.M17.Axis.NcToPlc <-> Outputs/ToPlc
//     PlcTask Outputs/Main.M17.Axis.PlcToNc <-> Inputs/FromPlc
//   kfe_rix_motion Instance <-> NC-Task 1 SAF/Axes/Axis 18 AT2K2-SOLID-MMS-02
//     PlcTask Inputs/Main.M18.Axis.NcToPlc <-> Outputs/ToPlc
//     PlcTask Outputs/Main.M18.Axis.PlcToNc <-> Inputs/FromPlc
//   kfe_rix_motion Instance <-> NC-Task 1 SAF/Axes/Axis 19 AT2K2-SOLID-MMS-03
//     PlcTask Inputs/Main.M19.Axis.NcToPlc <-> Outputs/ToPlc
//     PlcTask Outputs/Main.M19.Axis.PlcToNc <-> Inputs/FromPlc
//   kfe_rix_motion Instance <-> NC-Task 1 SAF/Axes/Axis 2 IM2K1-PPM-MMS
//     PlcTask Inputs/Main.M2.Axis.NcToPlc <-> Outputs/ToPlc
//     PlcTask Outputs/Main.M2.Axis.PlcToNc <-> Inputs/FromPlc
//   kfe_rix_motion Instance <-> NC-Task 1 SAF/Axes/Axis 20 AT2K2-SOLID-MMS-04
//     PlcTask Inputs/Main.M20.Axis.NcToPlc <-> Outputs/ToPlc
//     PlcTask Outputs/Main.M20.Axis.PlcToNc <-> Inputs/FromPlc
//   kfe_rix_motion Instance <-> NC-Task 1 SAF/Axes/Axis 21 LI3K2-K2B-MMS
//     PlcTask Inputs/Main.M21.Axis.NcToPlc <-> Outputs/ToPlc
//     PlcTask Outputs/Main.M21.Axis.PlcToNc <-> Inputs/FromPlc
//   kfe_rix_motion Instance <-> NC-Task 1 SAF/Axes/Axis 22 PF2K2-WFS-MMS-Y
//     PlcTask Inputs/Main.M22.Axis.NcToPlc <-> Outputs/ToPlc
//     PlcTask Outputs/Main.M22.Axis.PlcToNc <-> Inputs/FromPlc
//   kfe_rix_motion Instance <-> NC-Task 1 SAF/Axes/Axis 23 PF2K2-WFS-MMS-Z
//     PlcTask Inputs/Main.M23.Axis.NcToPlc <-> Outputs/ToPlc
//     PlcTask Outputs/Main.M23.Axis.PlcToNc <-> Inputs/FromPlc
//   kfe_rix_motion Instance <-> NC-Task 1 SAF/Axes/Axis 24 IM6K2-PPM-MMS
//     PlcTask Inputs/Main.M24.Axis.NcToPlc <-> Outputs/ToPlc
//     PlcTask Outputs/Main.M24.Axis.PlcToNc <-> Inputs/FromPlc
//   kfe_rix_motion Instance <-> NC-Task 1 SAF/Axes/Axis 25 AT1K2-SOLID-MMS-01
//     PlcTask Inputs/Main.M25.Axis.NcToPlc <-> Outputs/ToPlc
//     PlcTask Outputs/Main.M25.Axis.PlcToNc <-> Inputs/FromPlc
//   kfe_rix_motion Instance <-> NC-Task 1 SAF/Axes/Axis 26 AT1K2-SOLID-MMS-02
//     PlcTask Inputs/Main.M26.Axis.NcToPlc <-> Outputs/ToPlc
//     PlcTask Outputs/Main.M26.Axis.PlcToNc <-> Inputs/FromPlc
//   kfe_rix_motion Instance <-> NC-Task 1 SAF/Axes/Axis 27 AT1K2-SOLID-MMS-03
//     PlcTask Inputs/Main.M27.Axis.NcToPlc <-> Outputs/ToPlc
//     PlcTask Outputs/Main.M27.Axis.PlcToNc <-> Inputs/FromPlc
//   kfe_rix_motion Instance <-> NC-Task 1 SAF/Axes/Axis 28 SP1K2-PAX-FRAME-MMS-Y-01
//     PlcTask Inputs/Main.M28.Axis.NcToPlc <-> Outputs/ToPlc
//     PlcTask Outputs/Main.M28.Axis.PlcToNc <-> Inputs/FromPlc
//   kfe_rix_motion Instance <-> NC-Task 1 SAF/Axes/Axis 29 SP1K2-PAX-FRAME-MMS-Y-02
//     PlcTask Inputs/Main.M29.Axis.NcToPlc <-> Outputs/ToPlc
//     PlcTask Outputs/Main.M29.Axis.PlcToNc <-> Inputs/FromPlc
//   kfe_rix_motion Instance <-> NC-Task 1 SAF/Axes/Axis 3 SPARE
//     PlcTask Inputs/Main.M3.Axis.NcToPlc <-> Outputs/ToPlc
//     PlcTask Outputs/Main.M3.Axis.PlcToNc <-> Inputs/FromPlc
//   kfe_rix_motion Instance <-> NC-Task 1 SAF/Axes/Axis 30 SP1K2-PAX-FRAME-MMS-Y-03
//     PlcTask Inputs/Main.M30.Axis.NcToPlc <-> Outputs/ToPlc
//     PlcTask Outputs/Main.M30.Axis.PlcToNc <-> Inputs/FromPlc
//   kfe_rix_motion Instance <-> NC-Task 1 SAF/Axes/Axis 31 SP1K2-PAX-FRAME-MMS-X
//     PlcTask Inputs/Main.M31.Axis.NcToPlc <-> Outputs/ToPlc
//     PlcTask Outputs/Main.M31.Axis.PlcToNc <-> Inputs/FromPlc
//   kfe_rix_motion Instance <-> NC-Task 1 SAF/Axes/Axis 32 SP1K2-PAX-TAR-MMS-X
//     PlcTask Inputs/Main.M32.Axis.NcToPlc <-> Outputs/ToPlc
//     PlcTask Outputs/Main.M32.Axis.PlcToNc <-> Inputs/FromPlc
//   kfe_rix_motion Instance <-> NC-Task 1 SAF/Axes/Axis 33 SP1K2-PAX-TAR-MMS-Y
//     PlcTask Inputs/Main.M33.Axis.NcToPlc <-> Outputs/ToPlc
//     PlcTask Outputs/Main.M33.Axis.PlcToNc <-> Inputs/FromPlc
//   kfe_rix_motion Instance <-> NC-Task 1 SAF/Axes/Axis 34 SP1K2-PAX-TAR-MMS-Z
//     PlcTask Inputs/Main.M34.Axis.NcToPlc <-> Outputs/ToPlc
//     PlcTask Outputs/Main.M34.Axis.PlcToNc <-> Inputs/FromPlc
//   kfe_rix_motion Instance <-> NC-Task 1 SAF/Axes/Axis 35 SP1K2-PAX-TAR-MMS-RY
//     PlcTask Inputs/Main.M35.Axis.NcToPlc <-> Outputs/ToPlc
//     PlcTask Outputs/Main.M35.Axis.PlcToNc <-> Inputs/FromPlc
//   kfe_rix_motion Instance <-> NC-Task 1 SAF/Axes/Axis 36 SP1K2-PAX-BB-MMS-Y-01
//     PlcTask Inputs/Main.M36.Axis.NcToPlc <-> Outputs/ToPlc
//     PlcTask Outputs/Main.M36.Axis.PlcToNc <-> Inputs/FromPlc
//   kfe_rix_motion Instance <-> NC-Task 1 SAF/Axes/Axis 37 SP1K2-PAX-BB-MMS-Y-02
//     PlcTask Inputs/Main.M37.Axis.NcToPlc <-> Outputs/ToPlc
//     PlcTask Outputs/Main.M37.Axis.PlcToNc <-> Inputs/FromPlc
//   kfe_rix_motion Instance <-> NC-Task 1 SAF/Axes/Axis 38 SP2K2-TXAS-TAR-MMS-RX
//     PlcTask Inputs/Main.M38.Axis.NcToPlc <-> Outputs/ToPlc
//     PlcTask Outputs/Main.M38.Axis.PlcToNc <-> Inputs/FromPlc
//   kfe_rix_motion Instance <-> NC-Task 1 SAF/Axes/Axis 39 AT3K2-SOLID-MMS-Y-01
//     PlcTask Inputs/Main.M39.Axis.NcToPlc <-> Outputs/ToPlc
//     PlcTask Outputs/Main.M39.Axis.PlcToNc <-> Inputs/FromPlc
//   kfe_rix_motion Instance <-> NC-Task 1 SAF/Axes/Axis 4 IM1K2-PPM-MMS
//     PlcTask Inputs/Main.M4.Axis.NcToPlc <-> Outputs/ToPlc
//     PlcTask Outputs/Main.M4.Axis.PlcToNc <-> Inputs/FromPlc
//   kfe_rix_motion Instance <-> NC-Task 1 SAF/Axes/Axis 40 AT3K2-SOLID-MMS-Y-02
//     PlcTask Inputs/Main.M40.Axis.NcToPlc <-> Outputs/ToPlc
//     PlcTask Outputs/Main.M40.Axis.PlcToNc <-> Inputs/FromPlc
//   kfe_rix_motion Instance <-> NC-Task 1 SAF/Axes/Axis 5 AL1K2-L2SI-MMS
//     PlcTask Inputs/Main.M5.Axis.NcToPlc <-> Outputs/ToPlc
//     PlcTask Outputs/Main.M5.Axis.PlcToNc <-> Inputs/FromPlc
//   kfe_rix_motion Instance <-> NC-Task 1 SAF/Axes/Axis 6 IM2K2-PPM-MMS
//     PlcTask Inputs/Main.M6.Axis.NcToPlc <-> Outputs/ToPlc
//     PlcTask Outputs/Main.M6.Axis.PlcToNc <-> Inputs/FromPlc
//   kfe_rix_motion Instance <-> NC-Task 1 SAF/Axes/Axis 7 IM3K2-PPM-MMS
//     PlcTask Inputs/Main.M7.Axis.NcToPlc <-> Outputs/ToPlc
//     PlcTask Outputs/Main.M7.Axis.PlcToNc <-> Inputs/FromPlc
//   kfe_rix_motion Instance <-> NC-Task 1 SAF/Axes/Axis 8 IM4K2-PPM-MMS
//     PlcTask Inputs/Main.M8.Axis.NcToPlc <-> Outputs/ToPlc
//     PlcTask Outputs/Main.M8.Axis.PlcToNc <-> Inputs/FromPlc
//   kfe_rix_motion Instance <-> NC-Task 1 SAF/Axes/Axis 9 TM1K2-MMS-Y
//     PlcTask Inputs/Main.M9.Axis.NcToPlc <-> Outputs/ToPlc
//     PlcTask Outputs/Main.M9.Axis.PlcToNc <-> Inputs/FromPlc

CONFIGURATION kfe_rix_motion
    RESOURCE PLC ON TwinCAT3
        TASK PlcTask(INTERVAL := T#10ms, PRIORITY := 20);
        PROGRAM PRG_1_PlcTask WITH PlcTask : PRG_1_PlcTask;
    END_RESOURCE
END_CONFIGURATION

// ---- DUTs/DUT_SATT_Filter.TcDUT
TYPE DUT_SATT_Filter :
STRUCT
    {attribute 'pytmc' := '
        pv: MATERIAL
        io: input
        field: DESC Filter material name
    '}
    sFilterMaterial : STRING;

    {attribute 'pytmc' := '
        pv: THICKNESS
        io: input
        field: DESC Filter material thickness
        field: EGU um
    '}
    fFilterThickness_um : LREAL;
END_STRUCT
END_TYPE

// ---- DUTs/ENUM_SXR_SATT_Position.TcDUT
{attribute 'qualified_only'}
TYPE ENUM_SXR_SATT_Position :
(
    UNKNOWN := 0, // UNKNOWN must be in slot 0 or the FB breaks
    OUT := 1, // OUT at slot 1 is a convention
    FILTER1 := 2,
    FILTER2 := 3,
    FILTER3 := 4,
    FILTER4 := 5,
    FILTER5 := 6,
    FILTER6 := 7,
    FILTER7 := 8,
    FILTER8 := 9
);
END_TYPE

// ---- POUs/TM1K2/E_TM1K2_States.TcDUT
{attribute 'qualified_only'}
TYPE E_TM1K2_States :
// Adapted from E_ATM_States to add TARGET6
(
    Unknown := 0,
    OUT := 1,
    TARGET1 := 2,
    TARGET2 := 3,
    TARGET3 := 4,
    TARGET4 := 5,
    TARGET5 := 6,
    TARGET6 := 7,
    TARGET7 := 8,
    TARGET8 := 9
) UINT;
END_TYPE

// ---- POUs/TM2K2/E_TM2K2_States.TcDUT
{attribute 'qualified_only'}
TYPE E_TM2K2_States :
// Adapted from E_ATM_States to add TARGET6
(
    Unknown := 0,
    OUT := 1,
    TARGET1 := 2,
    TARGET2 := 3,
    TARGET3 := 4,
    TARGET4 := 5,
    TARGET5 := 6,
    TARGET6 := 7
) UINT;
END_TYPE

// ---- Version/Global_Version.TcGVL
{attribute 'TcGenerated'}
{attribute 'no-analysis'}
{attribute 'linkalways'}
// This function has been automatically generated from the project information.
VAR_GLOBAL CONSTANT
    {attribute 'const_non_replaced'}
    stLibVersion_plc_kfe_rix_motion : ST_LibVersion := (iMajor := 2, iMinor := 8, iBuild := 2, iRevision := 0, nFlags := 1, sVersion := '2.8.2');
END_VAR

// ---- GVLs/GVL.TcGVL

{attribute 'qualified_only'}
VAR_GLOBAL
    {attribute 'pytmc' := 'pv: PLC:RIX:MOTION:ARB:01'}
    fbArbiter1: FB_Arbiter(1);
    {attribute 'pytmc' := 'pv: PLC:RIX:MOTION:ARB:02'}
    fbArbiter2: FB_Arbiter(2);

    // For devices between the mirror and the stopper, uses 44 FF slots as of 1/12/2024, load 75 in EPICS (skip 125 for IOC load speed)
    {attribute 'pytmc' := '
        pv: PLC:RIX:MOTION:FFO:01
        astFF.array: 1..75
    '}
    {attribute 'TcLinkTo' := '.q_xFastFaultOut:=TIIB[PMPS_FFO]^Channel 1^Output'}
    fbFastFaultOutput1: FB_HardwareFFOutput := (bAutoReset := TRUE, i_sNetID:='172.21.42.126.1.1');

    // For devices after the stopper, uses 165 FF slots as of 1/12/2024, load all in EPICS
    {attribute 'pytmc' := '
        pv: PLC:RIX:MOTION:FFO:02
    '}
    {attribute 'TcLinkTo' := '.q_xFastFaultOut:=TIIB[PMPS_FFO]^Channel 2^Output'}
    fbFastFaultOutput2: FB_HardwareFFOutput := (bAutoReset := TRUE, i_sNetID:='172.21.42.126.1.1');

    //
     fbFastFaultOutput3: FB_HardwareFFOutput := (bAutoReset := TRUE, i_sNetID:='172.21.42.126.1.1');


    fbAtomicMass : FB_AtomicMass;
    fbAttenuatorElementDensity : FB_AttenuatorElementDensity;

    {attribute 'pytmc' := 'pv: PLC:RIX:MOTION:PMPS:ReqTrans'}
    rReqTrans AT %I*		: ARRAY [1..PMPS_GVL.AUX_ATTENUATORS] OF ST_PMPS_Attenuator_IO;
    {attribute 'pytmc' := 'pv: PLC:RIX:MOTION:PMPS:CurTrans'}
    rCurTrans AT %Q*		: ARRAY [1..PMPS_GVL.AUX_ATTENUATORS] OF ST_PMPS_Attenuator_IO;

    ePF1K2State: E_WFS_States;
    ePF2K2State: E_WFS_States;
END_VAR

VAR_GLOBAL CONSTANT
    iFiltersPerSATTBlade : INT := 8;
END_VAR

// ---- GVLs/Main.TcGVL
 {attribute 'qualified_only'}
VAR_GLOBAL
    // IM1K1-PPM-MMS
    {attribute 'pytmc' := 'pv: IM1K1:PPM:MMS'}
    {attribute 'TcLinkTo' := '.bLimitForwardEnable  := TIIB[IM1K1-EL7041]^STM Status^Status^Digital input 1;
                              .bLimitBackwardEnable := TIIB[IM1K1-EL7041]^STM Status^Status^Digital input 2;
                              .bBrakeRelease        := TIIB[IM1K1-EL2004]^Channel 1^Output'}
    M1: ST_MotionStage := (sName := 'IM1K1:PPM:MMS');

    // IM2K1-PPM-MMS
    {attribute 'pytmc' := 'pv: IM2K1:PPM:MMS'}
    {attribute 'TcLinkTo' := '.bLimitForwardEnable  := TIIB[IM2K1-EL7041]^STM Status^Status^Digital input 1;
                              .bLimitBackwardEnable := TIIB[IM2K1-EL7041]^STM Status^Status^Digital input 2;
                              .bBrakeRelease        := TIIB[IM2K1-EL2004]^Channel 1^Output'}
    M2: ST_MotionStage := (sName := 'IM2K1:PPM:MMS');

    // SPARE (Previously ZOS)
    M3: ST_MotionStage;

    // IM1K2-PPM-MMS
    {attribute 'pytmc' := 'pv: IM1K2:PPM:MMS'}
    {attribute 'TcLinkTo' := '.bLimitForwardEnable  := TIIB[IM1K2-EL7041-E1]^STM Status^Status^Digital input 1;
                              .bLimitBackwardEnable := TIIB[IM1K2-EL7041-E1]^STM Status^Status^Digital input 2;
                              .bBrakeRelease        := TIIB[IM1K2-EL2004-E3]^Channel 1^Output'}
    M4: ST_MotionStage := (sName := 'IM1K2:PPM:MMS');

    // AL1K2-L2SI: 1 Axis
    {attribute 'pytmc' := 'pv: AL1K2:L2SI:MMS'}
    {attribute 'TcLinkTo' := '.bLimitForwardEnable  := TIIB[AL1K2-EL7041-E1]^STM Status^Status^Digital input 1;
                              .bLimitBackwardEnable := TIIB[AL1K2-EL7041-E1]^STM Status^Status^Digital input 2;
                              .bBrakeRelease        := TIIB[AL1K2-EL2004-E3]^Channel 1^Output;
                              .nRawEncoderULINT     := TIIB[AL1K2-EL5042-E2]^FB Inputs Channel 1^Position'}
    M5: ST_MotionStage := (sName := 'AL1K2:L2SI:MMS');

    // IM2K2-PPM-MMS
    {attribute 'pytmc' := 'pv: IM2K2:PPM:MMS'}
    {attribute 'TcLinkTo' := '.bLimitForwardEnable  := TIIB[IM2K2-EL7041-E1]^STM Status^Status^Digital input 1;
                              .bLimitBackwardEnable := TIIB[IM2K2-EL7041-E1]^STM Status^Status^Digital input 2;
                              .bBrakeRelease        := TIIB[IM2K2-EL2004-E3]^Channel 1^Output'}
    M6: ST_MotionStage := (sName := 'IM2K2:PPM:MMS');

    // IM3K2-PPM-MMS
    {attribute 'pytmc' := 'pv: IM3K2:PPM:MMS'}
    {attribute 'TcLinkTo' := '.bLimitForwardEnable  := TIIB[IM3K2-EL7041-E1]^STM Status^Status^Digital input 1;
                              .bLimitBackwardEnable := TIIB[IM3K2-EL7041-E1]^STM Status^Status^Digital input 2;
                              .bBrakeRelease        := TIIB[IM3K2-EL2004-E3]^Channel 1^Output'}
    M7: ST_MotionStage := (sName := 'IM3K2:PPM:MMS');

    // IM4K2-PPM-MMS
    {attribute 'pytmc' := 'pv: IM4K2:PPM:MMS'}
    {attribute 'TcLinkTo' := '.bLimitForwardEnable  := TIIB[IM4K2-EL7041-E1]^STM Status^Status^Digital input 1;
                              .bLimitBackwardEnable := TIIB[IM4K2-EL7041-E1]^STM Status^Status^Digital input 2;
                              .bBrakeRelease        := TIIB[IM4K2-EL2004-E3]^Channel 1^Output'}
    M8: ST_MotionStage := (sName := 'IM4K2:PPM:MMS');

    // TM1K2: 2 Axes
    {attribute 'pytmc' := 'pv: TM1K2:ATM:MMS:Y'}
    {attribute 'TcLinkTo' := '.bLimitForwardEnable  := TIIB[TM1K2-EL7041-E1]^STM Status^Status^Digital input 1;
                              .bLimitBackwardEnable := TIIB[TM1K2-EL7041-E1]^STM Status^Status^Digital input 2;
                              .bBrakeRelease        := TIIB[TM1K2-EL2004-E4]^Channel 1^Output;
                              .nRawEncoderULINT     := TIIB[TM1K2-EL5042-E3]^FB Inputs Channel 1^Position'}
    M9: ST_MotionStage := (sName := 'TM1K2:ATM:MMS:Y');
    {attribute 'pytmc' := 'pv: TM1K2:ATM:MMS:X'}
    {attribute 'TcLinkTo' := '.nRawEncoderULINT     := TIIB[TM1K2-EL5042-E3]^FB Inputs Channel 2^Position'}
    M10: ST_MotionStage := (sName := 'TM1K2:ATM:MMS:X');

    // LI2K2-K2A_OUT: 1 Axis
    {attribute 'pytmc' := 'pv: LI2K2:K2A:MMS'}
    {attribute 'TcLinkTo' := '.bLimitForwardEnable  := TIIB[LI2K2-EL7041-E1]^STM Status^Status^Digital input 1;
                              .bLimitBackwardEnable := TIIB[LI2K2-EL7041-E1]^STM Status^Status^Digital input 2;
                              .bBrakeRelease        := TIIB[LI2K2-EL2004-E2]^Channel 1^Output;
                              .nRawEncoderULINT     := TIIB[LI2K2-EL5042-E3]^FB Inputs Channel 1^Position'}
    M11: ST_MotionStage := (sName := 'LI2K2:K2A:MMS');

    // PF1K2-WFS: 2 Axes
    {attribute 'pytmc' := 'pv: PF1K2:WFS:MMS:Y'}
    {attribute 'TcLinkTo' := '.bLimitForwardEnable  := TIIB[PF1K2-EL7041-E1]^STM Status^Status^Digital input 1;
                              .bLimitBackwardEnable := TIIB[PF1K2-EL7041-E1]^STM Status^Status^Digital input 2;
                              .bBrakeRelease        := TIIB[PF1K2-EL2004-E4]^Channel 1^Output;
                              .nRawEncoderULINT     := TIIB[PF1K2-EL5042-E3]^FB Inputs Channel 2^Position'}
    M12: ST_MotionStage := (sName := 'PF1K2:WFS:MMS:Y');
    {attribute 'pytmc' := 'pv: PF1K2:WFS:MMS:Z'}
    {attribute 'TcLinkTo' := '.nRawEncoderULINT     := TIIB[PF1K2-EL5042-E3]^FB Inputs Channel 1^Position'}
    M13: ST_MotionStage := (sName := 'PF1K2:WFS:MMS:Z');

    // IM5K2-PPM-MMS
    {attribute 'pytmc' := 'pv: IM5K2:PPM:MMS'}
    {attribute 'TcLinkTo' := '.bLimitForwardEnable  := TIIB[IM5K2-EL7041-E1]^STM Status^Status^Digital input 1;
                              .bLimitBackwardEnable := TIIB[IM5K2-EL7041-E1]^STM Status^Status^Digital input 2;
                              .bBrakeRelease        := TIIB[IM5K2-EL2004-E3]^Channel 1^Output'}
    M14: ST_MotionStage := (sName := 'IM5K2:PPM:MMS');

    // TM2K2: 2 Axes
    {attribute 'pytmc' := 'pv: TM2K2:ATM:MMS:Y'}
    {attribute 'TcLinkTo' := '.bLimitForwardEnable  := TIIB[TM2K2-EL7041-E1]^STM Status^Status^Digital input 1;
                              .bLimitBackwardEnable := TIIB[TM2K2-EL7041-E1]^STM Status^Status^Digital input 2;
                              .bBrakeRelease        := TIIB[TM2K2-EL2004-E4]^Channel 1^Output;
                              .nRawEncoderULINT     := TIIB[TM2K2-EL5042-E3]^FB Inputs Channel 1^Position'}
    M15: ST_MotionStage := (sName := 'TM2K2:ATM:MMS:Y');
    {attribute 'pytmc' := 'pv: TM2K2:ATM:MMS:X'}
    {attribute 'TcLinkTo' := '.nRawEncoderULINT     := TIIB[TM2K2-EL5042-E3]^FB Inputs Channel 2^Position'}
    M16: ST_MotionStage := (sName := 'TM2K2:ATM:MMS:X');

    //AT2K2: 4 Axes
(*

    AT2K2 Solid Attenuator notes (JJ-xray SN-11343)

    JJ    Label   EPICS    Stage     NC   Location

    1087      1   MMS:01   fbStage1  M17  Upstream-most
    1088      2   MMS:02   fbStage2  M18
    1086      3   MMS:03   fbStage3  M19
    1089      4   MMS:04   fbStage4  M20  Downstream-most

*)
    {attribute 'pytmc' := 'pv: AT2K2:L2SI:MMS:01'}
    {attribute 'TcLinkTo' := '
        .bLimitForwardEnable  := TIIB[AT2K2-EL7047-01]^STM Status^Status^Digital input 1;
        .bLimitBackwardEnable := TIIB[AT2K2-EL7047-01]^STM Status^Status^Digital input 2;
        .nRawEncoderULINT     := TIIB[AT2K2-EL5042-01]^FB Inputs Channel 1^Position
    '}
    M17: ST_MotionStage := (sName := 'AT2K2:L2SI:MMS:01');

    {attribute 'pytmc' := 'pv: AT2K2:L2SI:MMS:02'}
    {attribute 'TcLinkTo' := '
        .bLimitForwardEnable  := TIIB[AT2K2-EL7047-02]^STM Status^Status^Digital input 1;
        .bLimitBackwardEnable := TIIB[AT2K2-EL7047-02]^STM Status^Status^Digital input 2;
        .nRawEncoderULINT     := TIIB[AT2K2-EL5042-01]^FB Inputs Channel 2^Position
    '}
    M18: ST_MotionStage := (sName := 'AT2K2:L2SI:MMS:02');

    {attribute 'pytmc' := 'pv: AT2K2:L2SI:MMS:03'}
    {attribute 'TcLinkTo' := '
        .bLimitForwardEnable  := TIIB[AT2K2-EL7047-03]^STM Status^Status^Digital input 1;
        .bLimitBackwardEnable := TIIB[AT2K2-EL7047-03]^STM Status^Status^Digital input 2;
        .nRawEncoderULINT     := TIIB[AT2K2-EL5042-02]^FB Inputs Channel 1^Position
    '}
    M19: ST_MotionStage := (sName := 'AT2K2:L2SI:MMS:03');

    {attribute 'pytmc' := 'pv: AT2K2:L2SI:MMS:04'}
    {attribute 'TcLinkTo' := '
        .bLimitForwardEnable  := TIIB[AT2K2-EL7047-04]^STM Status^Status^Digital input 1;
        .bLimitBackwardEnable := TIIB[AT2K2-EL7047-04]^STM Status^Status^Digital input 2;
        .nRawEncoderULINT     := TIIB[AT2K2-EL5042-02]^FB Inputs Channel 2^Position
    '}
    M20: ST_MotionStage := (sName := 'AT2K2:L2SI:MMS:04');

    //LI3K2-K2B: 1 Axis
    {attribute 'pytmc' := 'pv: LI3K2:K2B:MMS'}
    {attribute 'TcLinkTo' := '.bLimitForwardEnable  := TIIB[LI3K2-EL7041-E1]^STM Status^Status^Digital input 1;
                              .bLimitBackwardEnable := TIIB[LI3K2-EL7041-E1]^STM Status^Status^Digital input 2;
                              .bBrakeRelease        := TIIB[LI3K2-EL2004-E3]^Channel 1^Output;
                              .nRawEncoderULINT     := TIIB[LI3K2-EL5042-E2]^FB Inputs Channel 1^Position'}
    M21: ST_MotionStage := (sName := 'LI3K2:K2B:MMS');

    //PF2K2: 2 Axes
    {attribute 'pytmc' := 'pv: PF2K2:WFS:MMS:Y'}
    {attribute 'TcLinkTo' := '.bLimitForwardEnable  := TIIB[PF2K2-EL7041-E1]^STM Status^Status^Digital input 1;
                              .bLimitBackwardEnable := TIIB[PF2K2-EL7041-E1]^STM Status^Status^Digital input 2;
                              .bBrakeRelease        := TIIB[PF2K2-EL2004-E4]^Channel 1^Output;
                              .nRawEncoderULINT     := TIIB[PF2K2-EL5042-E3]^FB Inputs Channel 2^Position'}
    M22: ST_MotionStage := (sName := 'PF2K2:WFS:MMS:Y');
    {attribute 'pytmc' := 'pv: PF2K2:WFS:MMS:Z'}
    {attribute 'TcLinkTo' := '.nRawEncoderULINT     := TIIB[PF2K2-EL5042-E3]^FB Inputs Channel 1^Position'}
    M23: ST_MotionStage := (sName := 'PF2K2:WFS:MMS:Z');


    //IM6K2: 1 Axis
    {attribute 'pytmc' := 'pv: IM6K2:PPM:MMS'}
    {attribute 'TcLinkTo' := '.bLimitForwardEnable  := TIIB[IM6K2-EL7041-E1]^STM Status^Status^Digital input 1;
                             .bLimitBackwardEnable := TIIB[IM6K2-EL7041-E1]^STM Status^Status^Digital input 2;
                             .bBrakeRelease        := TIIB[IM6K2-EL2004-E3]^Channel 1^Output'}
    M24: ST_MotionStage := (sName := 'IM6K2:PPM:MMS');


    //AT1K2: Blade 1


    {attribute 'pytmc' := 'pv: AT1K2:L2SI:MMS:01'}
    {attribute 'TcLinkTo' := '
        .bLimitForwardEnable  := TIIB[AT1K2-EL7047-01]^STM Status^Status^Digital input 1;
        .bLimitBackwardEnable := TIIB[AT1K2-EL7047-01]^STM Status^Status^Digital input 2;
        .nRawEncoderULINT     := TIIB[AT1K2-EL5042-01]^FB Inputs Channel 1^Position';
    ;}
    M25: ST_MotionStage := (sName := 'AT1K2:L2SI:MMS:01');

    //AT1K2: Blade 2

    {attribute 'pytmc' := 'pv: AT1K2:L2SI:MMS:02'}
    {attribute 'TcLinkTo' := '
        .bLimitForwardEnable  := TIIB[AT1K2-EL7047-02]^STM Status^Status^Digital input 1;
        .bLimitBackwardEnable := TIIB[AT1K2-EL7047-02]^STM Status^Status^Digital input 2;
        .nRawEncoderULINT     := TIIB[AT1K2-EL5042-01]^FB Inputs Channel 2^Position';
    ;}
    M26: ST_MotionStage := (sName := 'AT1K2:L2SI:MMS:02');

    //AT1K2: Mirror

    {attribute 'pytmc' := 'pv: AT1K2:L2SI:MMS:03'}
    {attribute 'TcLinkTo' := '
        .nRawEncoderULINT     := TIIB[AT1K2-EL5042-02]^FB Inputs Channel 1^Position';
    ;}
    M27: ST_MotionStage := (sName := 'AT1K2:L2SI:MMS:03');

    // PAX Motors
    {attribute 'pytmc' := 'pv: SP1K2:PAX:MMS:Y:01'}
    {attribute 'TcLinkTo' := '.bLimitForwardEnable  := TIIB[PAX-EL7047-E01]^STM Status^Status^Digital input 1;
                              .bLimitBackwardEnable := TIIB[PAX-EL7047-E01]^STM Status^Status^Digital input 2;
                              .nRawEncoderULINT     := TIIB[PAX-EL5042-E02]^FB Inputs Channel 1^Position'}
    M28: ST_MotionStage := (sName := 'SP1K2:PAX:FRAME:Y:01');

    {attribute 'pytmc' := 'pv: SP1K2:PAX:MMS:Y:02'}
    {attribute 'TcLinkTo' := '.bLimitForwardEnable  := TIIB[PAX-EL7047-E03]^STM Status^Status^Digital input 1;
                              .bLimitBackwardEnable := TIIB[PAX-EL7047-E03]^STM Status^Status^Digital input 2;
                              .nRawEncoderULINT     := TIIB[PAX-EL5042-E02]^FB Inputs Channel 2^Position'}

    M29: ST_MotionStage := (sName := 'SP1K2:PAX:FRAME:Y:02');

    {attribute 'pytmc' := 'pv: SP1K2:PAX:MMS:Y:03'}
    {attribute 'TcLinkTo' := '.bLimitForwardEnable  := TIIB[PAX-EL7047-E04]^STM Status^Status^Digital input 1;
                              .bLimitBackwardEnable := TIIB[PAX-EL7047-E04]^STM Status^Status^Digital input 2;
                              .nRawEncoderULINT     := TIIB[PAX-EL5042-E05]^FB Inputs Channel 1^Position'}
    M30: ST_MotionStage := (sName := 'SP1K2:PAX:FRAME:Y:03');

    {attribute 'pytmc' := 'pv: SP1K2:PAX:MMS:X:01'}
    {attribute 'TcLinkTo' := '.bLimitForwardEnable  := TIIB[PAX-EL7047-E06]^STM Status^Status^Digital input 2;
                              .bLimitBackwardEnable := TIIB[PAX-EL7047-E06]^STM Status^Status^Digital input 1;
                              .bBrakeRelease        := TIIB[PAX-EL2004-E07]^Channel 1^Output;
                              .nRawEncoderULINT     := TIIB[PAX-EL5042-E05]^FB Inputs Channel 2^Position'}
    M31: ST_MotionStage := (sName := 'SP1K2:PAX:FRAME:X');

    {attribute 'pytmc' := 'pv: SP1K2:PAX:MMS:X:02'}
    {attribute 'TcLinkTo' := '.bLimitForwardEnable  := TIID^PLC Rail (EtherCAT)^Power (EK1200)^Fiber Coupler (EK1521-0010)^Term 123 (EK1100)^Term 73 (EK1122)^PAX-DRL-02 (EK1100)^PAX-EL7047-E08^STM Status^Status^Digital input 2;
                              .bLimitBackwardEnable := TIID^PLC Rail (EtherCAT)^Power (EK1200)^Fiber Coupler (EK1521-0010)^Term 123 (EK1100)^Term 73 (EK1122)^PAX-DRL-02 (EK1100)^PAX-EL7047-E08^STM Status^Status^Digital input 1;
                              .nRawEncoderULINT     := TIID^PLC Rail (EtherCAT)^Power (EK1200)^Fiber Coupler (EK1521-0010)^Term 123 (EK1100)^Term 73 (EK1122)^PAX-DRL-02 (EK1100)^PAX-EL5042-E09^FB Inputs Channel 1^Position'}
    M32: ST_MotionStage := (sName := 'SP1K2:PAX:TAR:X');

    {attribute 'pytmc' := 'pv: SP1K2:PAX:MMS:Y:04'}
    {attribute 'TcLinkTo' := '.bLimitForwardEnable  := TIIB[PAX-EL7047-E10]^STM Status^Status^Digital input 2;
                              .bLimitBackwardEnable := TIIB[PAX-EL7047-E10]^STM Status^Status^Digital input 1;
                              .nRawEncoderULINT     := TIIB[PAX-EL5042-E09]^FB Inputs Channel 2^Position'}
    M33: ST_MotionStage := (sName := 'SP1K2:PAX:TAR:Y');

    {attribute 'pytmc' := 'pv: SP1K2:PAX:MMS:Z:01'}
    {attribute 'TcLinkTo' := '.bLimitForwardEnable  := TIIB[PAX-EL7047-E12]^STM Status^Status^Digital input 1;
                              .bLimitBackwardEnable := TIIB[PAX-EL7047-E12]^STM Status^Status^Digital input 2;
                              .nRawEncoderULINT     := TIIB[PAX-EL5042-E13]^FB Inputs Channel 1^Position'}
    M34: ST_MotionStage := (sName := 'SP1K2:PAX:TAR:Z');

    {attribute 'pytmc' := 'pv: SP1K2:PAX:MMS:RY:01'}
    {attribute 'TcLinkTo' := '.bLimitForwardEnable  := TIIB[PAX-EL7047-E14]^STM Status^Status^Digital input 1;
                              .bLimitBackwardEnable := TIIB[PAX-EL7047-E14]^STM Status^Status^Digital input 2;
                              .nRawEncoderULINT     := TIIB[PAX-EL5042-E13]^FB Inputs Channel 2^Position'}
    M35: ST_MotionStage := (sName := 'SP1K2:PAX:MMS:RY:01');

    {attribute 'pytmc' := 'pv: SP1K2:PAX:MMS:Y:05'}
    {attribute 'TcLinkTo' := '.bLimitForwardEnable  := TIIB[PAX-EL7047-E15]^STM Status^Status^Digital input 1;
                              .bLimitBackwardEnable := TIIB[PAX-EL7047-E15]^STM Status^Status^Digital input 2;
                              .nRawEncoderULINT     := TIIB[PAX-EL5042-E16]^FB Inputs Channel 1^Position'}
    M36: ST_MotionStage := (sName := 'SP1K2:PAX:BB:Y:01');

    {attribute 'pytmc' := 'pv: SP1K2:PAX:MMS:Y:06'}
    {attribute 'TcLinkTo' := '.bLimitForwardEnable  := TIIB[PAX-EL7047-E17]^STM Status^Status^Digital input 1;
                              .bLimitBackwardEnable := TIIB[PAX-EL7047-E17]^STM Status^Status^Digital input 2;
                              .nRawEncoderULINT     := TIIB[PAX-EL5042-E16]^FB Inputs Channel 2^Position'}
    M37: ST_MotionStage := (sName := 'SP1K2:PAX:BB:Y:02');


    // TXAS Motors
    {attribute 'pytmc' := 'pv: SP2K2:TXAS:MMS:RX:01'}
    {attribute 'TcLinkTo' := '.bLimitForwardEnable  := TIIB[K2S18-DRL-03-E7 (EL7047)]^STM Status^Status^Digital input 1;
                              .bLimitBackwardEnable := TIIB[K2S18-DRL-03-E7 (EL7047)]^STM Status^Status^Digital input 2;
                              .nRawEncoderULINT     := TIIB[K2S18-DRL-03-E8 (EL5112)]^ENC Status Channel 1^Counter value'}
    M38: ST_MotionStage := (sName := 'SP2K2:TXAS:MMS:RX:01');

    {attribute 'pytmc' := 'pv: AT3K2:L2SI:MMS:01'}
    {attribute 'TcLinkTo' := '.bLimitForwardEnable  := TIIB[K2S18-DRL-02-E6 (EL7047)]^STM Status^Status^Digital input 1;
                              .bLimitBackwardEnable := TIIB[K2S18-DRL-02-E6 (EL7047)]^STM Status^Status^Digital input 2;
                              .nRawEncoderULINT     := TIIB[K2S18-DRL-02-E5 (EL5042)]^FB Inputs Channel 2^Position'}
    M39: ST_MotionStage := (sName := 'AT3K2:SOLID:MMS:Y:01');

    {attribute 'pytmc' := 'pv: AT3K2:L2SI:MMS:02'}
    {attribute 'TcLinkTo' := '.bLimitForwardEnable  := TIIB[K2S18-DRL-02-E7 (EL7047)]^STM Status^Status^Digital input 1;
                              .bLimitBackwardEnable := TIIB[K2S18-DRL-02-E7 (EL7047)]^STM Status^Status^Digital input 2;
                              .nRawEncoderULINT     := TIIB[K2S18-DRL-02-E8 (EL5042)]^FB Inputs Channel 1^Position'}
    M40: ST_MotionStage := (sName := 'AT3K2:SOLID:MMS:Y:02');

    {attribute 'pytmc' := 'pv: SP2K2:TXAS:MMS:YAG:01'}
    {attribute 'TcLinkTo' := '.bLimitForwardEnable  := TIIB[K2S18-DRL-03-E13 (EL1124)]^Channel 1^Input;
                              .bLimitBackwardEnable := TIIB[K2S18-DRL-03-E13 (EL1124)]^Channel 2^Input;
                              .nRawEncoderULINT     := TIIB[K2S18-DRL-03-E9 (EL7037)]^ENC Status compact^Counter value'}
    M41: ST_MotionStage := (sName := 'SP2K2:TXAS:MMS:YAG:FOCUS');

END_VAR

// ---- POUs/PRG_1_PlcTask.TcPOU
PROGRAM PRG_1_PlcTask
VAR
    bDebug: BOOL := FALSE;
END_VAR

PRG_2_PMPS_PRE();

// Temporarily disable motors by setting bHardwareEnable to FALSE prior to running motion FB
//Main.M5.bHardwareEnable := bDebug;
//Main.M6.bHardwareEnable := bDebug;
//Main.M7.bHardwareEnable := bDebug;
//Main.M8.bHardwareEnable := bDebug;
//Main.M9.bHardwareEnable := bDebug;
//Main.M10.bHardwareEnable := bDebug;
//Main.M11.bHardwareEnable := bDebug;
//Main.M12.bHardwareEnable := bDebug;
//Main.M13.bHardwareEnable := bDebug;
//Main.M14.bHardwareEnable := bDebug;
//Main.M15.bHardwareEnable := bDebug;
//Main.M16.bHardwareEnable := bDebug;
// Note: AT2K2 has its own built-in debugging interface; see PRG_AT2K2_SOLID
// and its ``bDebug`` variable.

PRG_IM1K1_PPM();
PRG_IM2K1_PPM();
PRG_IM1K2_PPM();
PRG_AL1K2_L2SI();
PRG_IM2K2_PPM();
PRG_IM3K2_PPM();
PRG_IM4K2_PPM();
PRG_TM1K2_ATM();
PRG_LI2K2_K2A();
PRG_PF1K2_WFS();
PRG_IM5K2_PPM();
PRG_TM2K2_ATM();
PRG_AT1K2_SOLID();
PRG_AT2K2_SOLID();
PRG_LI3K2_K2B();
PRG_PF2K2_WFS();
PRG_IM6K2_PPM();

PRG_SP1K2_PAX();
PRG_SP2K2_TXAS();
PRG_AT3K2_SOLID();

PRG_3_PMPS_POST();
PRG_4_LOG();

END_PROGRAM

// ---- POUs/PRG_2_PMPS_PRE.TcPOU
PROGRAM PRG_2_PMPS_PRE
VAR
END_VAR

END_PROGRAM

// ---- POUs/PRG_IM1K1_PPM.TcPOU
PROGRAM PRG_IM1K1_PPM
VAR
    {attribute 'pytmc' := 'pv: IM1K1:PPM'}
    {attribute 'TcLinkTo' := '.fbGige.iIlluminatorINT := TIIB[IM1K1-EL4004]^AO Outputs Channel 1^Analog output;
                              .fbGige.bGigePower := TIIB[IM1K1-EL2004]^Channel 2^Output;
                              .fbPowerMeter.iVoltageINT := TIIB[IM1K1-EL3062]^AI Standard Channel 1^Value;
                              .fbPowerMeter.fbTempSensor.bError := TIIB[IM1K1-EL3314]^TC Inputs Channel 1^Status^Error;
                              .fbPowerMeter.fbTempSensor.bUnderrange := TIIB[IM1K1-EL3314]^TC Inputs Channel 1^Status^Underrange;
                              .fbPowerMeter.fbTempSensor.bOverrange := TIIB[IM1K1-EL3314]^TC Inputs Channel 1^Status^Overrange;
                              .fbPowerMeter.fbTempSensor.iRaw := TIIB[IM1K1-EL3314]^TC Inputs Channel 1^Value;
                              .fbYagTempSensor.bError := TIIB[IM1K1-EL3314]^TC Inputs Channel 2^Status^Error;
                              .fbYagTempSensor.bUnderrange := TIIB[IM1K1-EL3314]^TC Inputs Channel 2^Status^Underrange;
                              .fbYagTempSensor.bOverrange := TIIB[IM1K1-EL3314]^TC Inputs Channel 2^Status^Overrange;
                              .fbYagTempSensor.iRaw := TIIB[IM1K1-EL3314]^TC Inputs Channel 2^Value'}
    fbIM1K1: FB_PPM;

    fbStateSetup: FB_StateSetupHelper;
    stDefault: ST_PositionState := (
        fVelocity := 10,
        bMoveOk := TRUE,
        bValid := TRUE
    );
END_VAR


fbStateSetup(stPositionState:=stDefault, bSetDefault:=TRUE);

